// Set an alarm condition on the positive edge
IF (m_underRangeP.Q) THEN
	
	// Set underrange alarm TRUE
	Fault(fault:= f_FaultCode(TFaultPriority.Error, TFaultCondition.UnderRange), state:= TRUE);
	
END_IF
	
// Clear the alarm condition on a negative edge
IF (m_underRangeN.Q) THEN

	// Set underrange alarm FALSE
	Fault(fault:= f_FaultCode(TFaultPriority.Error, TFaultCondition.UnderRange), state:= FALSE);

END_IF

//
// Over range fault detection
//

// Use a TON delay timer
m_overRangeTON(IN:= channel.overRange);

// Rising Edge Trigger
m_overRangeP(CLK:= m_overRangeTON.Q);

// Falling Edge Trigger
m_overRangeN(CLK:= m_overRangeTON.Q);

// Set an alarm condition on the positive edge
IF (m_overRangeP.Q) THEN

	// Set overrange alarm TRUE
	Fault(fault:= f_FaultCode(TFaultPriority.Error, TFaultCondition.OverRange), state:= TRUE);
	
END_IF

// Clear the alarm condition on a negative edge
IF (m_overRangeN.Q) THEN

	// Set overrange alarm FALSE
	Fault(fault:= f_FaultCode(TFaultPriority.Error, TFaultCondition.OverRange), state:= FALSE);;
	
END_IF

//
// Short Circuit fault detection
//

// Use a TON delay timer
m_shortCircuitTON(IN:= channel.shortCircuit);

// Rising Edge Trigger
m_shortCircuitP(CLK:= m_shortCircuitTON.Q);

// Falling Edge Trigger
m_shortCircuitN(CLK:= m_shortCircuitTON.Q);

// Set an alarm condition on the positive edge
IF (m_shortCircuitP.Q) THEN

	// Set short circuit alarm TRUE
	Fault(fault:= f_FaultCode(TFaultPriority.Error, TFaultCondition.ShortCircuit), state:= TRUE);
	
END_IF

// Clear the alarm condition on a negative edge
IF (m_shortCircuitN.Q) THEN

	// Set short circuit alarm FALSE
	Fault(fault:= f_FaultCode(TFaultPriority.Error, TFaultCondition.ShortCircuit), state:= FALSE);;
	
END_IF

//
// Hardware error (wire break)
//

// Use a TON delay timer
m_errorTON(IN:= channel.error);

// Rising Edge Trigger
m_errorP(CLK:= m_errorTON.Q);

// Falling Edge Trigger
m_errorN(CLK:= m_errorTON.Q);

// Set an alarm condition on the positive edge
IF (m_errorP.Q) THEN

	// Set error alarm TRUE
	Fault(fault:= f_FaultCode(TFaultPriority.Error, TFaultCondition.HwError), state:= TRUE);
	m_WireBreakDetected := TRUE;
END_IF

// Clear the alarm condition on a negative edge
IF (m_errorN.Q) THEN

	// Set error alarm FALSE
	Fault(fault:= f_FaultCode(TFaultPriority.Error, TFaultCondition.HwError), state:= FALSE);
	m_WireBreakDetected := FALSE;
END_IF

IF (m_zeroCalEnable) THEN	

	// Calibration handling (zeroing) <TODO>
	m_zeroCalTimer();

	// Check if we are currently zeroing the transducer
	IF (m_zeroCalTimer.uliElapsedTime > 0) THEN

		// Update the data values
		m_zeroCalAccumulator := m_zeroCalAccumulator + m_filter.filteredValue;
		m_zeroCalCounter := m_zeroCalCounter + 1;

	ELSE

		// Done, calculate the average value
		IF (m_zeroCalCounter > 0) THEN

			m_rawVal := m_zeroCalAccumulator / m_zeroCalCounter;
	
		ELSE
	
			m_rawVal := m_filter.filteredValue;

		END_IF
		
		m_zeroCalRunning := FALSE;
		
	END_IF

ELSE
	
	// If no calibration is done set value to 0
	m_rawVal := 0;

END_IF

// Scale the raw calibration value to an output value
zeroCalValue := GetZeroCalValue();

(* ---------------------------------------------------------------------------
Func name   : 	AbortCal
Description : 	Aborts the calibration routine
Inputs      :	None
Returns     : 	None
Notes       : 	This routine will 0 out any previous output calibration value
--------------------------------------------------------------------------- *)

METHOD AbortCal
VAR_INPUT
END_VAR
m_zeroCalEnable := FALSE;
m_zeroCalAccumulator := 0.0;
m_zeroCalCounter := 0;
zeroCalValue := 0;
END_METHOD

(* ---------------------------------------------------------------------------
Func name   : 	Arm
Description : 	Enables all assiciated transducer alarms
Inputs      :	devId	-	device Id associated with the alarms in the system
Returns     : 	None
Notes       : 	The local alarm handler pointer is simply points to the
				global alarm handle function block.  Another approach could
				be to have any users of the analog transducer supply a
				fault handling routine with a common interface.
--------------------------------------------------------------------------- *)

METHOD Arm
VAR_INPUT
	devId		: UDeviceId;
END_VAR
// Set the local alarm handler pointer to the global handler so that the fault handler function can set alarms
m_pAlarmHandler := ADR(gAlarmHandler);

// Set the Device Id
m_devId := devId;
END_METHOD

(* ---------------------------------------------------------------------------
Func name   : 	Disarm
Description : 	Disables all assiciated transducer alarms
Inputs      :	None
Returns     : 	None
Notes       : 	This routine will also clear any active alarms before
				disabling the handler.
--------------------------------------------------------------------------- *)

METHOD Disarm
VAR_INPUT
END_VAR
// Clear any active alarms - Is this needed?
Fault(fault:= f_FaultCode(TFaultPriority.Error, TFaultCondition.UnderRange), state:= FALSE);
Fault(fault:= f_FaultCode(TFaultPriority.Error, TFaultCondition.OverRange), state:= FALSE);
Fault(fault:= f_FaultCode(TFaultPriority.Error, TFaultCondition.HwError), state:= FALSE);

// Clear the local alarm handler pointer - This will ignore all calls
m_pAlarmHandler := 0;
END_METHOD

(* ---------------------------------------------------------------------------
Func name   : 	Fault
Description : 	fault handling routine used as a common interface for
				setting/clearing transcuer faults.
Inputs      :	fault	-	fault code
				state	-	state of the fault
Returns     : 	None
Notes       : 	This routine assumes that when the transducer is armed,
				the alarm handler pointer will be non-zero, as well the
				internal m_devId parameter is set and valid.
--------------------------------------------------------------------------- *)

METHOD Fault
VAR_INPUT
	fault	: UFaultCode;
	state	: BOOL;
END_VAR
IF (m_pAlarmHandler <> 0) THEN
	
	IF (state) THEN
	
		m_pAlarmHandler^.Set(code:= f_AlarmCode(m_devId, fault));	
	
	ELSE
		
		m_pAlarmHandler^.Clear(code:= f_AlarmCode(m_devId, fault));	
	
	END_IF

END_IF
END_METHOD

(* ---------------------------------------------------------------------------
Func name   : 	FB_exit
Description : 	Destructor
Inputs      :	None
Returns     : 	None
Notes       : 	
--------------------------------------------------------------------------- *)

METHOD FB_exit : BOOL
VAR_INPUT
	bInCopyCode : BOOL; // if TRUE, the exit method is called for exiting an instance that is copied afterwards (online change)
END_VAR
// Do nothing
END_METHOD

(* ---------------------------------------------------------------------------
Func name   : 	FB_init
Description : 	Constructor
Inputs      :	iMinInput			:	minimum input
				iMaxInput			: 	maximum input
				rMinOutput			:	minimum output
				rMaxOutput			:	maximum output
				uiFilterSize 		:	Filter Sample Size
				uiFilterPrecision	:	Filter precision
				tDelay				:	Timer On Delay value
Returns     : 	None
Notes       : 	
--------------------------------------------------------------------------- *)

METHOD FB_init : BOOL
VAR_INPUT
	bInitRetains 				: BOOL; 		// if TRUE, the retain variables are initialized (warm start / cold start)
    bInCopyCode  				: BOOL; 		// if TRUE, the instance afterwards gets moved into the copy code (online change)
	iMinInput					: INT;			// minimum input
	iMaxInput					: INT;			// maximum input
	rMinOutput					: REAL;			// minimum output
	rMaxOutput					: REAL;			// maximum output
	uiFilterSize 				: UINT := 10;	// filter Sample Size
	uiFilterPrecision			: UINT := 4;	// filter precision
	tDelay						: TIME := T#1S;	// timer On Delay Value
END_VAR
// Set the member variables
m_iMinInput 	:= iMinInput;
m_iMaxInput		:= iMaxInput;
m_rMinOutput	:= rMinOutput;
m_rMaxOutput 	:= rMaxOutput;

// Initialize the calibration variables
m_zeroCalTimer.Initialize(msec:= 0, countDown:= TRUE, freeze:= FALSE);
m_zeroCalEnable := FALSE;
m_zeroCalRunning := FALSE;
m_zeroCalAccumulator := 0.0;
m_zeroCalCounter := 0;

// Initialize all of the timer delays
m_underRangeTON(PT:= tDelay);
m_overRangeTON(PT:= tDelay);
m_errorTON(PT:= tDelay);

// Initialize the Filter
// Set to default values here
m_filter.initialize(sampleSize:= uiFilterSize, precision:= uiFilterPrecision);

// Initialize the 'underrange', 'overrange', and 'error' positive edge detect signals
// to low so that we detect a positive edge if the signal is high at startup.
m_underRangeP(CLK:=FALSE);
m_overRangeP(CLK:=FALSE);
m_errorP(CLK:=FALSE);

// Initialize the output variables
signalValue := 0;
rawValue := 0;
zeroCalValue := 0;

// Set the local alarm handler pointer to the global handler
m_pAlarmHandler := ADR(gAlarmHandler);
END_METHOD

(* ---------------------------------------------------------------------------
Func name   : 	GetDevId
Description : 	Returns the transducer Device Id used for alarm categorization.
Inputs      :	None
Returns     : 	UDeviceId	-	Transducer device ID variable
Notes       : 	This function is currently used by the ENDP_Analog function block.
				I believe the End Point should set the Device Id instead of getting
				it from the transducer.  This could be a future improvement.
--------------------------------------------------------------------------- *)

METHOD GetDevId : UDeviceId
VAR_INPUT
END_VAR
GetDevId := m_devId;
END_METHOD

(* ---------------------------------------------------------------------------
Func name   : 	GetMaxOutput
Description : 	Returns the maximum output value of the transducer.
Inputs      :	None
Returns     : 	REAL	-	transducer maximum output value
Notes       : 	This routine is used by the fb_ENDP_Analog to get the
				transducer output limits.
--------------------------------------------------------------------------- *)

METHOD PUBLIC GetMaxOutput : REAL
VAR_INPUT
END_VAR
GetMaxOutput := m_rMaxOutput;
END_METHOD

(* ---------------------------------------------------------------------------
Func name   : 	GetMinOutput
Description : 	Returns the minimum output value of the transducer.
Inputs      :	None
Returns     : 	REAL	-	transducer minimum output value
Notes       : 	This routine is used by the fb_ENDP_Analog to get the
				transducer output limits.
--------------------------------------------------------------------------- *)

METHOD PUBLIC GetMinOutput : REAL
VAR_INPUT
END_VAR
GetMinOutput := m_rMinOutput;
END_METHOD

(* ---------------------------------------------------------------------------
Func name   : 	GetWireBreakStatus
Description : 	Returns the Status of a Wire Break Error.
Inputs      :	None
Returns     : 	BOOL- Status of Wire Break
Notes       : 	This method is used to get the status of the bool that reacts to a wire break.
--------------------------------------------------------------------------- *)
METHOD GetWireBreakStatus : BOOL
VAR_INPUT
END_VAR
GetWireBreakStatus := m_WireBreakDetected;
END_METHOD

(* ---------------------------------------------------------------------------
Func name   : 	GetZeroCalValue
Description : 	Scales and returns the current calibration value in mA.
Inputs      :	None
Returns     : 	REAL	-	scaled calibration value (mA)
Notes       : 	
--------------------------------------------------------------------------- *)

METHOD GetZeroCalValue : REAL
VAR_INPUT
END_VAR
// Scale the raw calibration value to an output value
 GetZeroCalValue := (m_rawVal * (m_rMaxOutput - m_rMinOutput) / (m_iMaxInput - m_iMinInput) + m_rMinOutput);
END_METHOD

(* ---------------------------------------------------------------------------
Func name   : 	InitAlarms
Description : 	Initializes the deviceId member variable used to set/clear
				the approproate alarms.
Inputs      :	devId	:	Device Id used for alarm integration
Returns     : 	None
Notes       : 	
--------------------------------------------------------------------------- *)

METHOD InitAlarms
VAR_INPUT
	devId		: UDeviceId;	// Device Id used for alarm integration
END_VAR
// Set the device id which is used for alarm integrtion
m_devId := devId;

// Register the handled alarm codes
m_pAlarmHandler^.RegisterAlarmCode(f_AlarmCode(m_devId, f_FaultCode(TFaultPriority.Error, TFaultCondition.UnderRange)));
m_pAlarmHandler^.RegisterAlarmCode(f_AlarmCode(m_devId, f_FaultCode(TFaultPriority.Error, TFaultCondition.OverRange)));
m_pAlarmHandler^.RegisterAlarmCode(f_AlarmCode(m_devId, f_FaultCode(TFaultPriority.Error, TFaultCondition.ShortCircuit)));
m_pAlarmHandler^.RegisterAlarmCode(f_AlarmCode(m_devId, f_FaultCode(TFaultPriority.Error, TFaultCondition.HwError)));
END_METHOD

(* ---------------------------------------------------------------------------
Func name   : 	IsZeroCalRunning
Description : 	Returns the status of the zero cal routine.
Inputs      :	None
Returns     : 	TRUE if zero cal running, FALSE otherwise
Notes       : 	
--------------------------------------------------------------------------- *)

METHOD IsZeroCalRunning : BOOL
VAR_INPUT
END_VAR
IsZeroCalRunning := m_zeroCalRunning;
END_METHOD

(* ---------------------------------------------------------------------------
Func name   : 	ZeroCal
Description : 	Averages the transducer signal input value to provide
				a calibration value reresenting a zero offset
Inputs      :	duration_ms	-	Duration of value averaging time in ms
Returns     : 	None
Notes       : 	This initializes the timer which runs the averaging routine
				in the main function block instantiation code.
--------------------------------------------------------------------------- *)

METHOD ZeroCal
VAR_INPUT
	duration_ms		: UINT;
END_VAR
// Initialize the data
m_zeroCalTimer.Initialize(msec := duration_ms, countDown := TRUE, freeze := FALSE);
m_zeroCalEnable := true;
m_zeroCalAccumulator := 0.0;
m_zeroCalCounter := 0;
zeroCalValue := 0;
m_zeroCalRunning := TRUE;
END_METHOD

END_FUNCTION_BLOCK

// 20 Program Organization Units/Input-Output Functions/fb_FreqTransducer
(*UPDATE: 			March. 18 2021 - Jaison Schaab

					Code Ported from Wago.
					
					Code has NOT Yet been tested.
*)

(*UPDATE: 			April. 28 2020 - Jaison Schaab

					Added the InitAlarms function which now NEEDS to be called in order to properly hook up the alarm monitors.
					This method is required because codesys does NOT properly propogate the FB_Init information like constructors
					in C code, so it is impossible to pass down the devceId information.
*)

FUNCTION_BLOCK fb_FreqTransducer
VAR_INPUT
	channel : Freq_ChannelInput; // will ~probably~ come from gstInputs. Ie HwRead + 2 copies already incurred. 
END_VAR
VAR_OUTPUT
	freqValue				: REAL;				// Scaled Signal Value (ex. mA or VDC)
	rawValue				: REAL;				// Raw Input Value (May be removed), no need to keep it UDINT, REAL is 3.4028e+38
END_VAR
VAR
	m_filter : fb_FilterExp;
	// these 2 are for Fault-handling. (hw-underrange, hw-overrange, hw-error) in this case. Which is not mapped like the Analog420input.
	m_devId : UDeviceId;
	m_pAlarmHandler : POINTER TO fb_AlarmHandler; // Alarm handler function pointer. NOTE_ Large Function. Expect this to be 1 Global func.
END_VAR

rawValue := DINT_TO_REAL(channel.value);
m_filter(inputValue:= (rawValue / 1000), filteredValue=> freqValue);

(* ---------------------------------------------------------------------------
Func name   : 	Fault
Description : 	fault handling routine used as a common interface for
				setting/clearing transcuer faults.
Inputs      :	fault	-	fault code
				state	-	state of the fault
Returns     : 	None
Notes       : 	This routine assumes that when the transducer is armed,
				the alarm handler pointer will be non-zero, as well the
				internal m_devId parameter is set and valid.
--------------------------------------------------------------------------- *)

METHOD FaultHandlerSetOrClear
VAR_INPUT
	fault	: UFaultCode;
	state	: BOOL;
END_VAR
IF (m_pAlarmHandler <> 0) THEN
	
	IF (state) THEN
	
		m_pAlarmHandler^.Set(code:= f_AlarmCode(m_devId, fault));	
	
	ELSE
		
		m_pAlarmHandler^.Clear(code:= f_AlarmCode(m_devId, fault));	
	
	END_IF

END_IF
END_METHOD

(* ---------------------------------------------------------------------------
Func name   : 	FB_init
Description : 	Constructor
Inputs      :	None
Returns     : 	None
Notes       : 	
--------------------------------------------------------------------------- *)

METHOD FB_init : BOOL
VAR_INPUT
	bInitRetains 		: BOOL; 		// if TRUE, the retain variables are initialized (warm start / cold start)
    bInCopyCode  		: BOOL; 		// if TRUE, the instance afterwards gets moved into the copy code (online change)
	histavgFiltSize: UINT;
	histavgFiltPrecision: UINT;
END_VAR
m_filter.initialize(sampleSize:= histavgFiltSize, precision:= histavgFiltPrecision);
freqValue := 0;
rawValue := 0;
END_METHOD

METHOD GetDevId : UDeviceId
VAR_INPUT
END_VAR
GetDevId := m_devId;
END_METHOD

(* ---------------------------------------------------------------------------
Func name   : 	InitAlarms
Description : 	Initializes the deviceId member variable used to set/clear
				the approproate alarms.
Inputs      :	devId	:	Device Id used for alarm integration
Returns     : 	None
Notes       : 	
--------------------------------------------------------------------------- *)

METHOD InitAlarms
VAR_INPUT
	devId : UDeviceId;
END_VAR
// Set the device id which is used for alarm integrtion
m_devId := devId;

// Register the handled alarm codes
// None Defined Yet <JAISON>
END_METHOD

END_FUNCTION_BLOCK

// 20 Program Organization Units/Instrument-Controller Functions/fb_Densitometer
(*AUTHOR:			Ryan Herdian*)
(*DATE:				June 16 / 2020*)
(*DESCRIPTION: 		This Function Block provides a BASE class for all densitometer objects.  The class
					consists of the following features:
					
						-	Min/Max configurable density ranges in specific gravity units whose range/values define the density units 
							of the entire class. Density is ratio agains clean water. Specific gravity of 1 is clean water.
						-	Raw density value in specific gravity units which is to be set by the derived class from its data source
						-	User settable unitless k-factor value which allows corrections in the desnsity value
						-	Corrected density value in density units which is the raw flow with k-factor applied
						-	Automatic k-factor calculation given known reference density in density units
					
					No Alarms are currently included, however alarm handler / fault function are defined.*)

(*NOTES:			The derived densitometer class is required to:
					
						- 	Set the m_densityMin/m_densityMax values in density unit [SGU].
							For example if the range of (0 - 1 [SGU]) then all values in that densitometer / denso instance
							 will return values in Specific Gravity Unit.  Including raw/corrected density.
						-	Set the m_rawDensity value in density units using the SetRawFlow() method.
						-	Initialize all values in the constructor including the user k-factor 
							and setting the alarm handler pointer.

*)

(*UPDATE: 			March. 18 2021 - Jaison Schaab

					Code Ported from Wago.
					
					Code has NOT Yet been tested.
*)

FUNCTION_BLOCK fb_Densitometer
VAR_INPUT
END_VAR
VAR_OUTPUT
END_VAR
VAR
	m_densityMin		: REAL			:= 0.0;			// in Specific Gravity Unit [SGU]
	m_densityMax		: REAL			:= 0.0;			// in [SGU]
	
	m_rawDensity		: REAL			:= 0.0;			// in density unit, e.g.: [SGU]
	
	m_userkfact			: REAL			:= 1.0;			// unitless multiplier (1.0 simply allows raw value output)
	
	// Fault Handling (Alarms)
	m_devId				: UDeviceId;					// Device Id used for alarm integration
END_VAR
VAR CONSTANT
	USER_K_FACTOR_MIN	: REAL := 0.1;					// minimum allowable user k-factor
	USER_K_FACTOR_MAX	: REAL := 10.0;					// maximum allowable user k-factor		
END_VAR

(* ---------------------------------------------------------------------------
Func name   : 	CalculateUserKFact
Description : 	Routine will calculate and set the densitometer k-factor
				so that the corrected density matches the input reference
				density value.
Inputs      :	refDensity	-	reference density value in density unit [SGU]
Returns     : 	None
Notes       : 	Use this routine to calibrate the densitometer to a known
				density in [SGU].
--------------------------------------------------------------------------- *)

METHOD CalculateUserkFact
VAR_INPUT
	refDensity	: REAL;		// reference density value in density unit [SGU]
END_VAR
IF (m_rawDensity > 0.0) THEN
	setUserKFact(kfact:= (refDensity / m_rawDensity) );
END_IF
END_METHOD

(* ---------------------------------------------------------------------------
Func name   : 	GetCorrectedDensitySGU
Description : 	Routine to calculate and return the corrected density
				with the user k-factor applied in density unit [SGU].
Inputs      :	None
Returns     : 	REAL	-	The corrected density value in density unit [SGU]
Notes       : 	
--------------------------------------------------------------------------- *)

METHOD GetCorrectedDensitySGU : REAL
VAR_INPUT
END_VAR
GetCorrectedDensitySGU	:= m_userkfact * m_rawDensity;
END_METHOD

(* ---------------------------------------------------------------------------
Func name   : 	GetDensityRange_MinMax
Description : 	Gets the minimum/maximum density range values from the densitometer
				in specific gravity units. Specific gravity of 1 is clean water.
Inputs      :	None
Returns     : 	minDensity		: 	denso minimum density value in density unit [SGU]
				maxDensity		:	denso maximum density value in density unit [SGU]
Notes       : 	
--------------------------------------------------------------------------- *)

METHOD GetDensityRange_MinMax
VAR_INPUT
END_VAR
VAR_OUTPUT
	minDensity		: REAL;		// minimum density value at transducer minimum value in [SGU]
	maxDensity		: REAL;		// maximum desnity value at transducer maximum value in [SGU]
END_VAR
// output the min/max density ranges
minDensity	:= m_densityMin;		// minimum density value at transducer minimum value in density unit [SGU]
maxDensity	:= m_densityMax;		// maximum desnity value at transducer maximum value in density unit [SGU]
END_METHOD

(* ---------------------------------------------------------------------------
Func name   : 	GetRawDensity
Description : 	Routine to return the raw density in density unit [SGU].
				This value does not have the k-factor applied.
Inputs      :	None
Returns     : 	REAL	-	The raw density value in Specific in density unit [SGU]
Notes       : 	
--------------------------------------------------------------------------- *)

METHOD GetRawDensity : REAL
VAR_INPUT
END_VAR
GetRawDensity	:= m_rawDensity;
END_METHOD

(* ---------------------------------------------------------------------------
Func name   : 	GetUserKFact
Description : 	Routine will return the unitless user k-factor value.
Inputs      :	None
Returns     : 	REAL	-	The unitless user k-factor value
Notes       : 	
--------------------------------------------------------------------------- *)

METHOD GetUserKFact : REAL
VAR_INPUT
END_VAR
GetUserKFact := m_userkfact;
END_METHOD

(* ---------------------------------------------------------------------------
Func name   : 	InitAlarms
Description : 	Initializes the deviceId member variable used to set/clear
				the approproate alarms.
Inputs      :	None
Returns     : 	None
Notes       : 	
--------------------------------------------------------------------------- *)

METHOD InitAlarms
VAR_INPUT
	devId		: UDeviceId;	// Device Id used for alarm integration
END_VAR
// Set the device id which is used for alarm integrtion
m_devId := devId;
END_METHOD

(* ---------------------------------------------------------------------------
Func name   : 	SetDensityRange_MinMax
Description : 	Sets the minimum/maximum desnity range values for the densitometer / denso
				in density unit Specific Gravity, [SGU].  The units defined by this range will
				define the units for all flow meter values.
Inputs      :	minDensity		: 	densitometer minimum flow value in density unit [SGU]
				maxDensity		:	densitometer maximum flow value in density unit [SGU]
Returns     : 	TRUE if min and max density are set. 
				FALSE if min and max density are not set (min density is greater than or equal to max density).
Notes       : 	All values in densitometer instance should be interpreted as 
				Specific Gravity, [SGU], including raw/corrected density.
--------------------------------------------------------------------------- *)

METHOD SetDensityRange_MinMax	: BOOL
VAR_INPUT
	minDensity		: REAL;		// minimum density value at transducer minimum value in density unit [SGU]
	maxDensity		: REAL;		// maximum density value at transducer maximum value in density unit [SGU]
END_VAR
IF (minDensity < maxDensity) THEN

	// Set the min/max densitometer range
	m_densityMin	:= minDensity;
	m_densityMax	:= maxDensity;
	
	SetDensityRange_MinMax	:= TRUE;

ELSE
	
	SetDensityRange_MinMax	:= FALSE;

END_IF
END_METHOD

(* ---------------------------------------------------------------------------
Func name   : 	SetRawDensity
Description : 	Private function which allows the derived classes to set the 
				densitometer rawDensity value in density unit [SGU].  
Inputs      :	density	-	Raw density in density unit [SGU]
Returns     : 	None
Notes       : 	The value will be limited by the initialized 
				minDensity/maxDensity values.
--------------------------------------------------------------------------- *)

METHOD PROTECTED SetRawDensity
VAR_INPUT
	density		: REAL;		// in density unit [SGU]
END_VAR
// Set the raw density value in the base densitometer class in density unit [SGU]
m_rawDensity	:= MAX(MIN(density, m_densityMax), m_densityMin);
END_METHOD

(* ---------------------------------------------------------------------------
Func name   : 	SetUserKFact
Description : 	Routine to set the unitless user k-factor value.
Inputs      :	kfact	-	The desried unitless user k-factor value
Returns     : 	None
Notes       : 	The value will be limited by the constants 
				USER_K_FACTOR_MIN and USER_K_FACTOR_MAX.
--------------------------------------------------------------------------- *)

METHOD setUserKFact
VAR_INPUT
	kfact	: REAL;
END_VAR
m_userkfact := MAX(MIN(kfact, USER_K_FACTOR_MAX), USER_K_FACTOR_MIN);
END_METHOD

END_FUNCTION_BLOCK

// 20 Program Organization Units/Instrument-Controller Functions/fb_ENDP_AnalogCalPressure
(*UPDATE: 			March. 18 2021 - Jaison Schaab

					Code Ported from Wago.
					
					Code has NOT Yet been tested.
*)

FUNCTION_BLOCK fb_ENDP_AnalogCalPressure
VAR_INPUT
	
END_VAR
VAR_OUTPUT
	correctedPressure 		: REAL;
	endpState				: INT;
END_VAR
VAR
	//Transducer Input
	m_pTransducer 	  		: POINTER TO fb_AnalogTransducer;
	
	//Config Variables - Need Get/Set Routines
	m_lowerCalPoint	  		: TCalibrationDataPoint; // m_inMin & m_outMin
	m_upperCalPoint	  		: TCalibrationDataPoint;//  m_inMax & m_outMax
	
	//Current configured pressure limits
	m_defaultPressMin 		: REAL := 0.0;
	m_defaultPressMax 		: REAL := 0.0;
	
	m_pressureMin		  		: REAL := 0.0; // physMin
	m_pressureMax		  		: REAL := 0.0; // physMax
	
	// Vars in fb_ENDP_Analog
	m_outDiffMultiplier 		: REAL;
	m_inDiffDivisor				: REAL; 
	m_offset					: REAL;
	m_hysteresis 				: REAL;
	
	m_rawPressure				: REAL := 0.0;
	m_userkfactor 				: REAL := 0.0;
	
	
	//Internal Status
	m_lowerCalTrigger 		: R_TRIG;
	m_upperCalTrigger 		: R_TRIG;
	
	m_calibrateLowPoint 	: BOOL;
	m_calibrateHighPoint 	: BOOL;
	// Handle Alarms
	m_devId 				: UDeviceId;
	LowAlarmMonitor			: fb_AlarmMonitor;
	LowWarningMonitor		: fb_AlarmMonitor;
	HighWarningMonitor		: fb_AlarmMonitor;
	HighAlarmMonitor		: fb_AlarmMonitor;
END_VAR

VAR CONSTANT
	USER_K_FACTOR_MAX 		: REAL := 10.0;
	USER_K_FACTOR_MIN 		: REAL := 1.0;
	DELAY_TON				: TIME := T#200MS;
END_VAR

// Ensure transducer pointer is not NULL
IF (m_pTransducer <> _NULL) THEN
	
	m_lowerCalTrigger(CLK:= (NOT m_pTransducer^.IsZeroCalRunning()) AND (m_calibrateLowPoint));
 	IF (m_lowerCalTrigger.Q) THEN
		m_lowerCalPoint.xValue	:= m_pTransducer^.GetZeroCalValue();
		
		m_calibrateLowPoint := FALSE;

		// Calculate a new minimum flow
		SetPressureRange(	minimum := f_LinearScale(value		:= m_pTransducer^.GetMinOutput(), 
															minInput	:= m_lowerCalPoint.xValue, 
															maxInput	:= m_upperCalPoint.xValue, 
															minOutput	:= m_lowerCalPoint.yValue, 
															maxOutput	:= m_upperCalPoint.yValue),
							maximum	:= m_pressureMax);
	END_IF
	
	m_upperCalTrigger(CLK:= (NOT m_pTransducer^.IsZeroCalRunning()) AND (m_calibrateHighPoint));
	IF (m_upperCalTrigger.Q) THEN
		m_upperCalPoint.xValue	:= m_pTransducer^.GetZeroCalValue();
		
		m_calibrateHighPoint := FALSE;
		
		// Calculate a new maximum pressure
		SetPressureRange(	minimum := m_pressureMin,
							maximum	:= f_LinearScale(value		:= m_pTransducer^.GetMaxOutput(), 
															minInput	:= m_lowerCalPoint.xValue, 
															maxInput	:= m_upperCalPoint.xValue, 
															minOutput	:= m_lowerCalPoint.yValue, 
															maxOutput	:= m_upperCalPoint.yValue));
	END_IF
	
	IF (NOT m_pTransducer^.IsZeroCalRunning()) THEN
		SetRawPressure( pressure := f_LinearScale(	value		:= m_pTransducer^.signalValue, 
															minInput	:= m_lowerCalPoint.xValue, 
															maxInput	:= m_upperCalPoint.xValue, 
															minOutput	:= m_lowerCalPoint.yValue, 
															maxOutput	:= m_upperCalPoint.yValue));
	END_IF							
ELSE
	SetRawPressure( pressure := 0.0);
END_IF

// Output the corrected pressure Value in kpa units
correctedPressure := GetCorrectedPressure();

//Monitor alarms.
LowAlarmMonitor.MonitorReal(correctedPressure);
LowWarningMonitor.MonitorReal(correctedPressure);
HighWarningMonitor.MonitorReal(correctedPressure);
HighAlarmMonitor.MonitorReal(correctedPressure);

IF (m_pTransducer^.channel.error) THEN
	endpState := TEnuHmiGaugeState.LowAlarm;
ELSIF(LowAlarmMonitor.GetState()) THEN
	endpState := TEnuHmiGaugeState.LowAlarm;
ELSIF(HighWarningMonitor.GetState()) THEN
	endpState := TO_INT(TEnuHmiGaugeState.HighWarning);
ELSIF(LowWarningMonitor.GetState()) THEN
	endpState := TEnuHmiGaugeState.LowWarning;
ELSE
	endpState := TEnuHmiGaugeState.No_Alarm;			
END_IF

(* ---------------------------------------------------------------------------
Func name   : 	CalculateUserKFact
Description : 	
Inputs      :	
Returns     : 	None
Notes       : 	
--------------------------------------------------------------------------- *)

METHOD CalculateUserKFactor
VAR_INPUT
	refPress	: REAL;
END_VAR
IF (m_rawPressure > 0.0) THEN
	SetUserKFactor(refPress  / m_rawPressure);
END_IF
END_METHOD

(* ---------------------------------------------------------------------------
Func name   : 	CalibrateHighDataPoint
Description : 	Averages the transducer signal input value to provide
				a high calibration data point for the flowmeter scale.
Inputs      :	val			-	Calibration value in Kpa units
				duration_ms	-	Duration of value averaging time in ms
Returns     : 	None
Notes       : 	
--------------------------------------------------------------------------- *)

METHOD CalibrateHighDataPoint
VAR_INPUT
	val				: REAL;		// Calibration value in volume/t units
	duration_ms 	: UINT;		// Duration of value averaging time in ms
END_VAR
IF ((NOT m_calibrateLowPoint) AND (NOT m_calibrateHighPoint)) THEN
	m_pTransducer^.ZeroCal(duration_ms:= duration_ms);
	m_upperCalPoint.yValue	:= val;
	m_calibrateHighPoint := TRUE;
END_IF
END_METHOD

(* ---------------------------------------------------------------------------
Func name   : 	CalibrateLowDataPoint
Description : 	Averages the transducer signal input value to provide
				a low calibration data point for the flowmeter scale.
Inputs      :	val			-	Calibration value in volume/t units
				duration_ms	-	Duration of value averaging time in ms
Returns     : 	None
Notes       : 	
--------------------------------------------------------------------------- *)

METHOD CalibrateLowDataPoint
VAR_INPUT
	val				: REAL;		// Calibration value in volume/t units
	duration_ms 	: UINT;		// Duration of value averaging time in ms
END_VAR
VAR
	minFlow		: REAL;
	maxFlow		: REAL;
END_VAR
IF ((NOT m_calibrateLowPoint) AND (NOT m_calibrateHighPoint)) THEN
	m_pTransducer^.ZeroCal(duration_ms:= duration_ms);
	m_lowerCalPoint.yValue	:= val;
	m_calibrateLowPoint := TRUE;
END_IF
END_METHOD

(* ---------------------------------------------------------------------------
Func name   : 	ClearCalibration
Description : 	Clears all calibration of the pressure transducer and resets to
				the default constructor scale.
Inputs      :	None
Returns     : 	None
Notes       : 	
--------------------------------------------------------------------------- *)

METHOD ClearCalibration
VAR_INPUT
END_VAR
// Reset to default values
m_lowerCalPoint.xValue	:= m_pTransducer^.GetMinOutput();
m_lowerCalPoint.yValue	:= m_defaultPressMin;

m_upperCalPoint.xValue	:= m_pTransducer^.GetMaxOutput();
m_upperCalPoint.yValue	:= m_defaultPressMax;

SetPressureRange(minimum := m_defaultPressMin,maximum := m_defaultPressMax);
						
m_calibrateLowPoint		:= FALSE;
m_calibrateHighPoint	:= FALSE;
END_METHOD

(* ---------------------------------------------------------------------------
Func name   : 	FB_exit
Description : 	Destructor
Inputs      :	None
Returns     : 	None
Notes       : 	
--------------------------------------------------------------------------- *)

METHOD FB_exit : BOOL
VAR_INPUT
	bInCopyCode : BOOL; // if TRUE, the exit method is called for exiting an instance that is copied afterwards (online change)
END_VAR
// Do nothing
END_METHOD

METHOD FB_Init
VAR_INPUT
	bInitRetains 	: BOOL;
	bInCopyCode  	: BOOL;
	
	pTransducer  	: POINTER TO fb_AnalogTransducer;
	minPress	 	: REAL;
	maxPress	 	: REAL;
	perctHysteresis : REAL;
END_VAR
// Default User K-Factor to 1.0
SetUserKFactor( k := 1.0);

// Default the raw press value to 0
SetRawPressure( pressure := 0.0);

// Set the pressure ranges in pascals
m_defaultPressMin := minPress;
m_defaultPressMax := maxPress;

SetPressureRange( minimum := minPress, maximum := maxPress);

// Set the transducer pointer
m_pTransducer := pTransducer;

// Initialize the calibration values
m_lowerCalPoint.xValue := m_pTransducer^.GetMinOutput(); //inMin
m_lowerCalPoint.yValue := minPress; //outMin

m_upperCalPoint.xValue := m_pTransducer^.GetMaxOutput(); // inMax
m_upperCalPoint.yValue := maxPress; // outMax

m_outDiffMultiplier    := m_upperCalPoint.yValue - m_lowerCalPoint.yValue;
m_inDiffDivisor		   := m_upperCalPoint.xValue - m_upperCalPoint.xValue;

IF( m_inDiffDivisor = 0.0) THEN
	m_inDiffDivisor := 0.000001; //protect against div-by-0, only ONCE, and produce VERY-LARGE Bad value.
                                  //Beckhoff-tcNov was doing this A.every cycle and B.returned 0.0 if Bad, which is normal value. hard to notice.
END_IF


m_hysteresis := perctHysteresis / 100;
m_lowerCalTrigger(CLK := FALSE);
m_upperCalTrigger(CLK := FALSE);

m_calibrateLowPoint 	:= FALSE;
m_calibrateHighPoint 	:= FALSE;
END_METHOD

(* ---------------------------------------------------------------------------
Func name   : 	GetConfigData
Description : 	equivalent of "Configure" bkhff-legacy-names.
				
Inputs      :	2-end-range-values, 1 offset, 4 alarms - 7 values.
				state	-	state of the fault
Returns     : 	None
Notes       : 	
--------------------------------------------------------------------------- *)

METHOD GetConfigData
VAR_INPUT
	//cfg : TEndpAnalogCfg;
MinValue : REAL;
MaxValue : REAL;
OffsetValue : REAL;
LowLimit : REAL;
LowWarning : REAL;
HighWarning : REAL;
HighLimit : REAL;
END_VAR
m_lowerCalPoint.yValue := MinValue;
m_upperCalPoint.yValue := MaxValue;
m_offset := OffsetValue;

//LowAlarmMonitor.m_limit.limitOn := LowLimit;
LowAlarmMonitor.SetLimitReal(LowLimit, LowLimit*(1 + m_hysteresis)); // + 0.5);

//LowWarningMonitor.m_limit.limitOn := LowWarning;
LowWarningMonitor.SetLimitReal(LowWarning, LowWarning*(1 + m_hysteresis)); // + 0.5);

//HighWarningMonitor.m_limit.limitOn := HighWarning;
HighWarningMonitor.SetLimitReal(HighWarning, HighWarning*(1 - m_hysteresis)); // - 0.5);

//HighAlarmMonitor.m_limit.limitOn := HighLimit;
HighAlarmMonitor.SetLimitReal(HighLimit, HighLimit*(1 - m_hysteresis)); // - 0.5);
END_METHOD

METHOD GetCorrectedPressure : REAL
VAR_INPUT
END_VAR
GetCorrectedPressure := m_userkfactor * m_rawPressure;
END_METHOD

(* ---------------------------------------------------------------------------
Func name   : 	GetLowerCalDataPoint
Description : 	returns the flowmeter lower calibration data point.
Inputs      :	None
Returns     : 	REAL	-	lower calibration data point
Notes       : 	
--------------------------------------------------------------------------- *)

METHOD GetLowerCalDataPoint : TCalibrationDataPoint
VAR_INPUT
END_VAR
GetLowerCalDataPoint := m_lowerCalPoint;
END_METHOD

(* ---------------------------------------------------------------------------
Func name   : 	GetPressureRange
Description : 	Gets the minimum/maximum pressure range values from the pressure transducer
				in volume/t units.
Inputs      :	None
Returns     : 	minPressure		: 	Pressure Transducer's minimum pressure value (kpa)
				maxPressure		:	Pressure Transducer's maximum pressure value (kpa)
Notes       : 	
--------------------------------------------------------------------------- *)

METHOD GetPressureRange
VAR_INPUT
END_VAR
VAR_OUTPUT
	minPressure : REAL;	// minimum pressure value at transducer's minimum value (kpa)
	maxPressure : REAL; // maximum pressure value at transducer's maximum value (kpa)
END_VAR
minPressure := m_pressureMin;
maxPressure := m_pressureMax;
END_METHOD

(* ---------------------------------------------------------------------------
Func name   : 	GetRawPressure
Description : 	Routine to return the raw pressure value in Kpa units.
				This value does not have the k-factor applied.
Inputs      :	None
Returns     : 	REAL	-	The raw pressure value in Kpa
Notes       : 	
--------------------------------------------------------------------------- *)

METHOD GetRawPressure : REAL
VAR_INPUT
END_VAR
GetRawPressure := m_rawPressure;
END_METHOD

(* ---------------------------------------------------------------------------
Func name   : 	GetUpperCalDataPoint
Description : 	returns the flowmeter upper calibration data point.
Inputs      :	None
Returns     : 	REAL	-	upper calibration data point
Notes       : 	
--------------------------------------------------------------------------- *)

METHOD GetUpperCalDataPoint : TCalibrationDataPoint
VAR_INPUT
END_VAR
GetUpperCalDataPoint := m_upperCalPoint;
END_METHOD

METHOD GetUserAlarms
VAR_OUTPUT
	outLAlarm 	:REAL;
	outLWarn 	:REAL;
	outHWarn 	:REAL;
	outHAlarm 	:REAL;
END_VAR
outLAlarm 	:= LREAL_TO_REAL(LowAlarmMonitor.m_limit.limitOn);
outLWarn  	:= LREAL_TO_REAL(LowWarningMonitor.m_limit.limitOn);
outHWarn 	:= LREAL_TO_REAL(HighWarningMonitor.m_limit.limitOn);
outHAlarm 	:= LREAL_TO_REAL(HighAlarmMonitor.m_limit.limitOn);
END_METHOD

(* ---------------------------------------------------------------------------
Func name   : 	GetUserKFactor
Description : 	Routine will return the unitless user k-factor value.
Inputs      :	None
Returns     : 	REAL	-	The unitless user k-factor value
Notes       : 	
--------------------------------------------------------------------------- *)

METHOD GetUserKFactor : REAL
VAR_INPUT
END_VAR
GetUserKFactor := m_userkfactor;
END_METHOD

(* ---------------------------------------------------------------------------
Func name   : 	InitAlarms
Description : 	Initializes the deviceId member variable used to set/clear
				the approproate alarms.
Inputs      :	None
Returns     : 	None
Notes       : 	
--------------------------------------------------------------------------- *)

METHOD InitAlarms
VAR_INPUT
END_VAR
// Set the device id which is used for alarm integration
m_devId := m_pTransducer^.GetDevId();

LowAlarmMonitor.InitAlarm(f_AlarmCode(m_devId, f_FaultCode(TFaultPriority.Warning, TFaultCondition.UnderLimit)), TAlarmMonitorType.lower_limit, DELAY_TON);
LowWarningMonitor.InitAlarm(f_AlarmCode(m_devId, f_FaultCode(TFaultPriority.Warning, TFaultCondition.UnderWarning)), TAlarmMonitorType.lower_limit, DELAY_TON);
HighWarningMonitor.InitAlarm(f_AlarmCode(m_devId, f_FaultCode(TFaultPriority.Warning, TFaultCondition.OverWarning)), TAlarmMonitorType.upper_limit, DELAY_TON);
HighAlarmMonitor.InitAlarm(f_AlarmCode(m_devId, f_FaultCode(TFaultPriority.Warning, TFaultCondition.OverLimit)), TAlarmMonitorType.upper_limit, DELAY_TON);
END_METHOD

METHOD SetHysteresis
VAR_INPUT
	perctHysteresis : REAL;
END_VAR
m_hysteresis := perctHysteresis/100;
END_METHOD

(* ---------------------------------------------------------------------------
Func name   : 	SetLowerCalDataPoint
Description : 	sets the flowmeter lower calibration data point.
Inputs      :	calPoint	-	calibration data point
Returns     : 	None
Notes       : 	
--------------------------------------------------------------------------- *)

METHOD SetLowerCalDataPoint
VAR_INPUT
	calPoint	: TCalibrationDataPoint;
END_VAR
m_lowerCalPoint := calPoint;
END_METHOD

METHOD SetPressureRange : BOOL
VAR_INPUT
	minimum : REAL;
	maximum : REAL;
END_VAR
IF ( maximum > minimum) THEN
	m_pressureMin := minimum;
	m_pressureMax := maximum;
	SetPressureRange := TRUE;
ELSE
	SetPressureRange := FALSE;
END_IF
END_METHOD

METHOD SetRangeUserAlarms
VAR_INPUT
	loAlarm : REAL;
	loWarn  : REAL;
	hiWarn  : REAL;
	hiAlarm : REAL;
END_VAR
IF (NOTUSED = loAlarm OR NOTUSED_LOMAX = loAlarm OR loAlarm < m_lowerCalPoint.yValue OR loAlarm > m_upperCalPoint.yValue) THEN
	loAlarm := NOTUSED_LOMAX;
	LowAlarmMonitor.DisableLimit();
ELSE
	LowAlarmMonitor.EnableLimit();
END_IF
LowAlarmMonitor.SetLimitReal(loAlarm, (loAlarm  + MAX(0.001, ABS(loAlarm)) * m_hysteresis));

IF (NOTUSED = loWarn OR loWarn <= loAlarm OR loAlarm > m_upperCalPoint.yValue ) THEN
	loWarn := loAlarm;
	LowWarningMonitor.DisableLimit();
ELSE
	LowWarningMonitor.EnableLimit();
END_IF
LowWarningMonitor.SetLimitReal(loWarn, (loWarn  + MAX(0.001, ABS(loWarn)) * m_hysteresis));

IF (NOTUSED = hiAlarm OR NOTUSED_HIMAX = hiAlarm OR hiAlarm < m_lowerCalPoint.yValue OR hiAlarm > m_upperCalPoint.yValue) THEN
	hiAlarm := NOTUSED_HIMAX; //Guaranteed greater than m_outMax; We pick _some_ large value.
	HighAlarmMonitor.DisableLimit();
ELSE
	HighAlarmMonitor.EnableLimit();
END_IF
HighAlarmMonitor.SetLimitReal(hiAlarm, (hiAlarm - MAX(0.001, ABS(hiAlarm)) * m_hysteresis));

IF (NOTUSED = hiWarn OR hiWarn >= hiAlarm OR hiWarn < m_lowerCalPoint.yValue) THEN
	hiWarn := hiAlarm;   //User doesnt have ability to set these individually. So WE define this order. So hiAlarm - already set.
	HighWarningMonitor.DisableLimit();
ELSE
	HighWarningMonitor.EnableLimit();
END_IF
HighWarningMonitor.SetLimitReal(hiWarn, (hiWarn - MAX(0.001, ABS(hiWarn)) * m_hysteresis));
END_METHOD

METHOD SetRawPressure : REAL
VAR_INPUT
	pressure : REAL;
END_VAR
m_rawPressure := MAX(MIN(pressure,m_pressureMax), m_pressureMin);

SetRawPressure := m_rawPressure;
END_METHOD

(* ---------------------------------------------------------------------------
Func name   : 	SetUpperCalDataPoint
Description : 	sets the flowmeter upper calibration data point.
Inputs      :	calPoint	-	calibration data point
Returns     : 	None
Notes       : 	
--------------------------------------------------------------------------- *)

METHOD SetUpperCalDataPoint
VAR_INPUT
	calPoint	: TCalibrationDataPoint;
END_VAR
m_upperCalPoint := calPoint;
END_METHOD

METHOD SetUserKFactor
VAR_INPUT
	k : REAL;
END_VAR
m_userkfactor := MAX(MIN(k, USER_K_FACTOR_MAX), USER_K_FACTOR_MIN);
END_METHOD

END_FUNCTION_BLOCK

// 20 Program Organization Units/Instrument-Controller Functions/fb_ENDP_AnalogDensitometer
(*AUTHOR:			Ryan Herdian*)
(*DATE:				June 17, 2020*)
(*DESCRIPTION: 		Derived densitometer class which provides an analog denso object.  The raw density
					value is obtained from the configured "Analog Transducer" object in the configured
					density unit, Specific Gravity Unit [SGU].*)

(*UPDATE: 			March. 18 2021 - Jaison Schaab

					Code Ported from Wago.
					
					Code has NOT Yet been tested.
*)

FUNCTION_BLOCK fb_ENDP_AnalogDensitometer EXTENDS fb_Densitometer
VAR_INPUT
END_VAR
VAR_OUTPUT
	correctedDensity	: REAL;								// Corrected density in density unit Specific Gravity Unit, [SGU]
END_VAR
VAR
	// Transducer input
	m_pTransducer	 	: POINTER TO fb_AnalogTransducer;	// Pointer to transducer
END_VAR

// Ensure transducer pointer is not NULL
IF (m_pTransducer <> _NULL) THEN

	// Set the raw density value in the base densitometer class in density unit, e.g.: Specific Gravity Unit, [SGU]
	SetRawDensity(density:= f_LinearScale(	value		:= m_pTransducer^.signalValue, 
											minInput	:= m_pTransducer^.GetMinOutput(), 
											maxInput	:= m_pTransducer^.GetMaxOutput(), 
											minOutput	:= m_densityMin, 
											maxOutput	:= m_densityMax));
													
ELSE
	SetRawDensity(density:= 0.0);

END_IF
							
// Output the corrected Flow Value in voume/t units
correctedDensity := GetCorrectedDensitySGU();

(* ---------------------------------------------------------------------------
Func name   : 	FB_exit
Description : 	Destructor
Inputs      :	None
Returns     : 	None
Notes       : 	
--------------------------------------------------------------------------- *)

METHOD FB_exit : BOOL
VAR_INPUT
	bInCopyCode : BOOL; // if TRUE, the exit method is called for exiting an instance that is copied afterwards (online change)
END_VAR
// Do Nothing
END_METHOD

(* ---------------------------------------------------------------------------
Func name   : 	FB_init
Description : 	Constructor
Inputs      :	pTransducer			:	transducer pointer
				minDensity			: 	minimum density value at transducer minimum value in density unit, e.g.: Specific Gravity Unit, [SGU]
				maxDensity			:	maximum density value at transducer maximum value in density unit, e.g.: Specific Gravity Unit, [SGU]
Returns     : 	None
Notes       : 	
--------------------------------------------------------------------------- *)

METHOD FB_init : BOOL
VAR_INPUT
	bInitRetains 		: BOOL; 							// if TRUE, the retain variables are initialized (warm start / cold start)
    bInCopyCode  		: BOOL; 							// if TRUE, the instance afterwards gets moved into the copy code (online change)
	pTransducer 		: POINTER TO fb_AnalogTransducer;	// transducer pointer
	minDensity 			: REAL;								// minimum Density value at transducer minimum value in density unit, e.g.: Specific Gravity Unit, [SGU]
	maxDensity 			: REAL;								// maximum Density value at transducer maximum value in density unit, e.g.: Specific Gravity Unit, [SGU]
END_VAR
// Default User kFact to 1.0
SetUserKFact(kfact := 1.0);

// Default the raw density value to 0
SetRawDensity(density:= 0.0);

// Set the density ranges in density unit, e.g.: Specific Gravity Unit, [SGU]
SetDensityRange_MinMax(	minDensity	:= minDensity, 
						maxDensity	:= maxDensity);

// Set the transducer pointer
m_pTransducer := pTransducer;
END_METHOD

END_FUNCTION_BLOCK

// 20 Program Organization Units/Instrument-Controller Functions/fb_ENDP_AnalogFlowmeter
(*AUTHOR:			Jaison Schaab*)
(*DATE:				June 9 / 2020*)
(*DESCRIPTION: 		Derived flow meter class which provides an analog flow meter object.  The raw volume flow
					value is obtained from the configured "Analog Transducer" object in the configured
					 volume/t units.*)

(*UPDATE: 			March. 23 2021 - Jaison Schaab

					Code Is fully tested and functional.				
*)
					 
(*UPDATE: 			March. 18 2021 - Jaison Schaab

					Code Ported from Wago.
					
					Code has NOT Yet been tested.
*)
					 
(*UPDATE: 			August. 31 2020 - Jaison Schaab

					Added new calibration data points to define the analog flow meter scaling.  These data points can
					be reset to the constructor values using the "ClearCalibration" routine.  They are set using the
					"CalibrateHighDataPoint" and "CalibrateLowDataPoint" or by simply writing them via the "SetLowerCalDataPoint"
					and "SetUpperCalDataPoint".
					
					Keep in mind that these values will need to be added to the config memory space in order to retain them.
*)	
					 
(*UPDATE: 			June. 23 2020 - Jaison Schaab

					Removed backdoor (m_pAlarmHandler : POINTER TO fb_AlarmHandler) alarm handler function pointer
					in order to simplify the alarm system.  Any alarms at this level should define a instance
					of the fb_AlarmMonitor class which will handle the alarm registration/set/clear.
*)					 				 

FUNCTION_BLOCK fb_ENDP_AnalogFlowmeter EXTENDS fb_FlowMeter
VAR_INPUT
END_VAR
VAR_OUTPUT
	correctedFlow				: REAL;								// Corrected flow in volume/t units
END_VAR
VAR
	// Transducer input
	m_pTransducer				: POINTER TO fb_AnalogTransducer;	// Pointer to transducer
	
	// Config Variables - Need Get/Set Routines
	m_lowerCalPoint				: TCalibrationDataPoint;			// Lower calibration data point
	m_upperCalPoint				: TCalibrationDataPoint;			// Upper calibration data point
	
	
	// Internal Status
	m_lowerCalTrigger			: R_TRIG;
	m_upperCalTrigger			: R_TRIG;
	
	m_calibrateLowPoint			: BOOL;
	m_calibrateHighPoint		: BOOL;

END_VAR

// Ensure transducer pointer is not NULL
IF (m_pTransducer <> _NULL) THEN
	
	m_lowerCalTrigger(CLK:= (NOT m_pTransducer^.IsZeroCalRunning()) AND (m_calibrateLowPoint));
 	IF (m_lowerCalTrigger.Q) THEN
		m_lowerCalPoint.xValue	:= m_pTransducer^.GetZeroCalValue();
		
		m_calibrateLowPoint := FALSE;

		// Calculate a new minimum flow
		SetFlowRange_MinMax(	minFlow := f_LinearScale(	value		:= m_pTransducer^.GetMinOutput(), 
															minInput	:= m_lowerCalPoint.xValue, 
															maxInput	:= m_upperCalPoint.xValue, 
															minOutput	:= m_lowerCalPoint.yValue, 
															maxOutput	:= m_upperCalPoint.yValue),
								maxFlow	:= m_flowMax);
	END_IF
	
	m_upperCalTrigger(CLK:= (NOT m_pTransducer^.IsZeroCalRunning()) AND (m_calibrateHighPoint));
	IF (m_upperCalTrigger.Q) THEN
		m_upperCalPoint.xValue	:= m_pTransducer^.GetZeroCalValue();
		
		m_calibrateHighPoint := FALSE;
		
		// Calculate a new maximum flow
		SetFlowRange_MinMax(	minFlow := m_flowMin,
								maxFlow	:= f_LinearScale(	value		:= m_pTransducer^.GetMaxOutput(), 
															minInput	:= m_lowerCalPoint.xValue, 
															maxInput	:= m_upperCalPoint.xValue, 
															minOutput	:= m_lowerCalPoint.yValue, 
															maxOutput	:= m_upperCalPoint.yValue));
	END_IF
	
	// Set the raw flow value in the base flow meter class in volume/t units
	//SetRawFlow(flow:= f_LinearScale(	value		:= m_pTransducer^.signalValue, 
	//									minInput	:= m_pTransducer^.GetMinOutput(), 
	//									maxInput	:= m_pTransducer^.GetMaxOutput(), 
	//									minOutput	:= m_flowMin, 
	//									maxOutput	:= m_flowMax);
	IF (NOT m_pTransducer^.IsZeroCalRunning()) THEN
		SetRawFlow(flow:= f_LinearScale(	value		:= m_pTransducer^.signalValue, 
											minInput	:= m_lowerCalPoint.xValue, 
											maxInput	:= m_upperCalPoint.xValue, 
											minOutput	:= m_lowerCalPoint.yValue, 
											maxOutput	:= m_upperCalPoint.yValue));
	END_IF
								
ELSE

	SetRawFlow(flow:= 0.0);

END_IF
						
// Output the corrected Flow Value in voume/t units
correctedFlow := GetCorrectedFlow();

// Update the totalizers in voume/t units
m_totalizer1(	inputRate	:= MAX(0, GetCorrectedFlow()), 
				totalValue	=> m_total1);
				
m_totalizer2(	inputRate	:= MAX(0, GetCorrectedFlow()), 
				totalValue	=> m_total2);
				
m_totalizer3(	inputRate	:= MAX(0, GetCorrectedFlow()), 
				totalValue	=> m_total3);
				
// Update Alarms
m_LowFlowLimitAlarm.MonitorReal(	value	:= correctedFlow);
m_LowFlowWarningAlarm.MonitorReal(	value	:= correctedFlow);
m_HighFlowWarningAlarm.MonitorReal(	value	:= correctedFlow);
m_HighFlowLimitAlarm.MonitorReal(	value	:= correctedFlow);

(* ---------------------------------------------------------------------------
Func name   : 	CalibrateHighDataPoint
Description : 	Averages the transducer signal input value to provide
				a high calibration data point for the flowmeter scale.
Inputs      :	val			-	Calibration value in volume/t units
				duration_ms	-	Duration of value averaging time in ms
Returns     : 	None
Notes       : 	
--------------------------------------------------------------------------- *)

METHOD CalibrateHighDataPoint
VAR_INPUT
	val				: REAL;		// Calibration value in volume/t units
	duration_ms 	: UINT;		// Duration of value averaging time in ms
END_VAR
IF ((NOT m_calibrateLowPoint) AND (NOT m_calibrateHighPoint)) THEN
	m_pTransducer^.ZeroCal(duration_ms:= duration_ms);
	m_upperCalPoint.yValue	:= val;
	m_calibrateHighPoint := TRUE;
END_IF
END_METHOD

(* ---------------------------------------------------------------------------
Func name   : 	CalibrateLowDataPoint
Description : 	Averages the transducer signal input value to provide
				a low calibration data point for the flowmeter scale.
Inputs      :	val			-	Calibration value in volume/t units
				duration_ms	-	Duration of value averaging time in ms
Returns     : 	None
Notes       : 	
--------------------------------------------------------------------------- *)

METHOD CalibrateLowDataPoint
VAR_INPUT
	val				: REAL;		// Calibration value in volume/t units
	duration_ms 	: UINT;		// Duration of value averaging time in ms
END_VAR
VAR
	minFlow		: REAL;
	maxFlow		: REAL;
END_VAR
IF ((NOT m_calibrateLowPoint) AND (NOT m_calibrateHighPoint)) THEN
	m_pTransducer^.ZeroCal(duration_ms:= duration_ms);
	m_lowerCalPoint.yValue	:= val;
	m_calibrateLowPoint := TRUE;
END_IF
END_METHOD

(* ---------------------------------------------------------------------------
Func name   : 	ClearCalibration
Description : 	Clears all calibration of the flowmeter and resets to
				the default constructor scale.
Inputs      :	None
Returns     : 	None
Notes       : 	
--------------------------------------------------------------------------- *)

METHOD ClearCalibration
VAR_INPUT
END_VAR
// Reset to default values
m_lowerCalPoint.xValue	:= m_pTransducer^.GetMinOutput();
m_lowerCalPoint.yValue	:= m_defaultFlowMin;

m_upperCalPoint.xValue	:= m_pTransducer^.GetMaxOutput();
m_upperCalPoint.yValue	:= m_defaultFlowMax;

SetFlowRange_MinMax(	minFlow := m_defaultFlowMin,
						maxFlow	:= m_defaultFlowMax);
						
m_calibrateLowPoint		:= FALSE;
m_calibrateHighPoint	:= FALSE;
END_METHOD

(* ---------------------------------------------------------------------------
Func name   : 	FB_exit
Description : 	Destructor
Inputs      :	None
Returns     : 	None
Notes       : 	
--------------------------------------------------------------------------- *)

METHOD FB_exit : BOOL
VAR_INPUT
	bInCopyCode : BOOL; // if TRUE, the exit method is called for exiting an instance that is copied afterwards (online change)
END_VAR
// Do nothing
END_METHOD

(* ---------------------------------------------------------------------------
Func name   : 	FB_init
Description : 	Constructor
Inputs      :	pTransducer			:	transducer pointer
				minFlow				: 	minimum flow value at transducer minimum value (volume/t)
				maxFlow				:	maximum flow value at transducer maximum value (volume/t)
Returns     : 	None
Notes       : 	
--------------------------------------------------------------------------- *)

METHOD FB_init : BOOL
VAR_INPUT
	bInitRetains 		: BOOL; 							// if TRUE, the retain variables are initialized (warm start / cold start)
    bInCopyCode  		: BOOL; 							// if TRUE, the instance afterwards gets moved into the copy code (online change)
	pTransducer 		: POINTER TO fb_AnalogTransducer;	// transducer pointer
	minFlow 			: REAL;								// minimum flow value at transducer minimum value (volume/t)
	maxFlow 			: REAL;								// maximum flow value at transducer maximum value (volume/t)
END_VAR
// Default User kFact to 1.0
SetUserKFact(kfact := 1.0);

// Default the raw flow value to 0
SetRawFlow(flow:= 0.0);

// Initialize / Reset the totalizers
m_totalizer1.Reset();
m_totalizer2.Reset();
m_totalizer1.Reset();

// Enable the totalizers as default
m_totalizer1.Enable();
m_totalizer2.Enable();
m_totalizer3.Enable();

// Set the flow ranges in volume/t units
m_defaultFlowMin		:= minFlow;				// in volume/t units
m_defaultFlowMax 		:= maxFlow;				// in volume/t units
SetFlowRange_MinMax(	minFlow := minFlow,
						maxFlow	:= maxFlow);
						
// Set the transducer pointer
m_pTransducer := pTransducer;

// Initialize the calibration values
m_lowerCalPoint.xValue	:= m_pTransducer^.GetMinOutput();
m_lowerCalPoint.yValue	:= minFlow;

m_upperCalPoint.xValue	:= m_pTransducer^.GetMaxOutput();
m_upperCalPoint.yValue	:= maxFlow;


m_lowerCalTrigger(CLK:= FALSE);
m_upperCalTrigger(CLK:= FALSE);
m_calibrateLowPoint		:= FALSE;
m_calibrateHighPoint	:= FALSE;
END_METHOD

(* ---------------------------------------------------------------------------
Func name   : 	GetLowerCalDataPoint
Description : 	returns the flowmeter lower calibration data point.
Inputs      :	None
Returns     : 	REAL	-	lower calibration data point
Notes       : 	
--------------------------------------------------------------------------- *)

METHOD GetLowerCalDataPoint : TCalibrationDataPoint
VAR_INPUT
END_VAR
GetLowerCalDataPoint := m_lowerCalPoint;
END_METHOD

(* ---------------------------------------------------------------------------
Func name   : 	GetUpperCalDataPoint
Description : 	returns the flowmeter upper calibration data point.
Inputs      :	None
Returns     : 	REAL	-	upper calibration data point
Notes       : 	
--------------------------------------------------------------------------- *)

METHOD GetUpperCalDataPoint : TCalibrationDataPoint
VAR_INPUT
END_VAR
GetUpperCalDataPoint := m_upperCalPoint;
END_METHOD

(* ---------------------------------------------------------------------------
Func name   : 	SetLowerCalDataPoint
Description : 	sets the flowmeter lower calibration data point.
Inputs      :	calPoint	-	calibration data point
Returns     : 	None
Notes       : 	
--------------------------------------------------------------------------- *)

METHOD SetLowerCalDataPoint
VAR_INPUT
	calPoint	: TCalibrationDataPoint;
END_VAR
m_lowerCalPoint := calPoint;
END_METHOD

(* ---------------------------------------------------------------------------
Func name   : 	SetUpperCalDataPoint
Description : 	sets the flowmeter upper calibration data point.
Inputs      :	calPoint	-	calibration data point
Returns     : 	None
Notes       : 	
--------------------------------------------------------------------------- *)

METHOD SetUpperCalDataPoint
VAR_INPUT
	calPoint	: TCalibrationDataPoint;
END_VAR
m_upperCalPoint := calPoint;
END_METHOD

END_FUNCTION_BLOCK

// 20 Program Organization Units/Instrument-Controller Functions/fb_FlowMeter
(*AUTHOR:			Jaison Schaab*)
(*DATE:				June 9 / 2020*)
(*DESCRIPTION: 		This Function Block provides a BASE class for all flow meter objects.  The class
					consists of the following features:
					
						-	Min/Max configurable flow ranges in volume/t units whose range/values define the flow units of the entire class
						-	Raw volume flow value in volume/t units which is to be set by the derived class from its data source
						-	User settable unitless k-factor value which allows corrections in the flow value
						-	Corrected volume flow value in volume/t units which is the raw flow with k-factor applied
						-	Automatic k-factor calculation given known reference flow in volume/t units
						-	3 seperate volume flow totalizers with pause/resume/reset functionality
					
					No Alarms are currently included. however alarm handler / fault function are defined.*)

(*UPDATE: 			March. 23 2021 - Jaison Schaab

					Code Is fully tested and functional.				
*)

(*UPDATE: 			March. 18 2021 - Jaison Schaab

					Code Ported from Wago.
					
					Code has NOT Yet been tested.
*)

(*UPDATE: 			August. 31 2020 - Jaison Schaab

					Added "m_defaultFlowMin" and "m_defaultFlowMax" values which will allow the flow meter range
					to be re-defined through calibration and then restored to orginal constructor limits.
*)	

(*UPDATE: 			June. 23 2020 - Jaison Schaab

					Removed backdoor (m_pAlarmHandler : POINTER TO fb_AlarmHandler) alarm handler function pointer
					in order to simplify the alarm system.  Any alarms at this level should define a instance
					of the fb_AlarmMonitor class which will handle the alarm registration/set/clear.
*)	

(*NOTES:			The derived flow meter class is required to:
					
						- 	Define and set the m_flowMin/m_flowMax values in the desired volume flow units.
							For example if the range of (0 - 10 m3/min) then all values in that flowmeter instance
							 will return values in m3/min.  Including raw/corrected flow and all totalizers.
						-	Set the m_rawFlow value in volume/t units using the SetRawFlow() method.
						-	cyclically call the 3 totalizer objects to ensure they are updated on each scan.
						-	Initialize all values in the constructor including the user k-factor, totalizer
							reset/enable, and setting the alarm handler pointer.

*)

FUNCTION_BLOCK fb_FlowMeter
VAR_INPUT
END_VAR
VAR_OUTPUT
END_VAR
VAR
	// Default constructor flow limits
	m_defaultFlowMin		: REAL			:= 0.0;			// in volume/t units
	m_defaultFlowMax 		: REAL			:= 0.0;			// in volume/t units	
	
	// Current configured flow limits
	m_flowMin				: REAL			:= 0.0;			// in volume/t units
	m_flowMax 				: REAL			:= 0.0;			// in volume/t units	

	m_rawFlow				: REAL			:= 0.0;			// in volume/t units

	// Config Variables
	m_userkfact				: REAL			:= 1.0;			// unitless multiplier (1.0 simply allows raw value output)
	
	m_total1				: REAL			:= 0.0;			// in volume/t units
	m_total2				: REAL			:= 0.0;			// in volume/t units
	m_total3				: REAL			:= 0.0;			// in volume/t units
	
	m_totalizer1			: Totalizer;					// totalizer 1
	m_totalizer2			: Totalizer;					// totalizer 2
	m_totalizer3			: Totalizer;					// totalizer 3
	
	// Fault Handling (Alarms)
	m_devId					: UDeviceId;					// Device Id used for alarm integration
	
	// Alarms
	m_LowFlowLimitAlarm 	: fb_AlarmMonitor;				// Alarm - Low flow limit alarm
	m_LowFlowWarningAlarm 	: fb_AlarmMonitor;				// Alarm - Low flow warning alarm
	m_HighFlowWarningAlarm 	: fb_AlarmMonitor;				// Alarm - high flow warning alarm
	m_HighFlowLimitAlarm 	: fb_AlarmMonitor;				// Alarm - high flow limit alarm
	
END_VAR
VAR CONSTANT
	USER_K_FACTOR_MIN		: REAL := 0.1;					// minimum allowable user k-factor
	USER_K_FACTOR_MAX		: REAL := 10.0;					// maximum allowable user k-factor
	ALARM_HYST_PERCENT		: REAL := 1.0;					// hysteresis percentage for reseting alarms
END_VAR

(* ---------------------------------------------------------------------------
Func name   : 	CalculateUserKFact
Description : 	Routine will calculate and set the flow meter k-factor
				so that the corrected flow matches the input reference
				flow value.
Inputs      :	refFlow	-	reference flow value in volume/t
Returns     : 	None
Notes       : 	Use this routine to calibrate the flow meter to a known
				flow in volume/t.
--------------------------------------------------------------------------- *)

METHOD CalculateUserKFact
VAR_INPUT
	refFlow	: REAL;
END_VAR
IF (m_rawFlow > 0.0) THEN
	SetUserKFact(refFlow / m_rawFlow);
END_IF
END_METHOD

(* ---------------------------------------------------------------------------
Func name   : 	GetCorrectedFlow
Description : 	Routine to calculate and return the corrected volume flow
				with the user k-factor applied in volume/t units.
Inputs      :	None
Returns     : 	REAL	-	The corrected volume flow value in volume/t
Notes       : 	
--------------------------------------------------------------------------- *)

METHOD GetCorrectedFlow : REAL
VAR_INPUT
END_VAR
GetCorrectedFlow := m_userkfact * m_rawFlow;
END_METHOD

(* ---------------------------------------------------------------------------
Func name   : 	GetFlowRange_MinMax
Description : 	Gets the minimum/maximum flow range values from the flowmeter
				in volume/t units.
Inputs      :	None
Returns     : 	minFlow		: 	flowmeter minimum flow value (volume/t)
				maxFlow		:	flowmeter maximum flow value (volume/t)
Notes       : 	
--------------------------------------------------------------------------- *)

METHOD GetFlowRange_MinMax
VAR_INPUT
END_VAR
VAR_OUTPUT
	minFlow 	: REAL;		// minimum flow value at transducer minimum value (volume/t)
	maxFlow 	: REAL;		// maximum flow value at transducer maximum value (volume/t)
END_VAR
// output the min/max flowmeter ranges
minFlow := m_flowMin;
maxFlow := m_flowMax;
END_METHOD

(* ---------------------------------------------------------------------------
Func name   : 	GetRawFlow
Description : 	Routine to return the raw volume flow value in volume/t units.
				This value does not have the k-factor applied.
Inputs      :	None
Returns     : 	REAL	-	The raw volume flow value in volume/t
Notes       : 	
--------------------------------------------------------------------------- *)

METHOD GetRawFlow : REAL
VAR_INPUT
END_VAR
GetRawFlow := m_rawFlow;
END_METHOD

(* ---------------------------------------------------------------------------
Func name   : 	GetUserAlarms
Description : 	Gets the low/high flow warning alarm value in volume/t units.
Inputs      :	None
Returns     : 	lowFlowWarn		: 	low flow warning alarm value (volume/t)
				highFlowWarn	:	high flow warning alarm value (volume/t)
Notes       : 	
--------------------------------------------------------------------------- *)

METHOD GetUserAlarms
VAR_INPUT
END_VAR
VAR_OUTPUT
	lowFlowWarn 	: REAL;		// low flow warning alarm value (volume/t)
	highFlowWarn	: REAL;		// high flow warning alarm value (volume/t)
END_VAR
lowFlowWarn  	:= LREAL_TO_REAL(m_LowFlowWarningAlarm.m_limit.limitOn);
highFlowWarn  	:= LREAL_TO_REAL(m_HighFlowWarningAlarm.m_limit.limitOn);
END_METHOD

(* ---------------------------------------------------------------------------
Func name   : 	GetUserKFact
Description : 	Routine will return the unitless user k-factor value.
Inputs      :	None
Returns     : 	REAL	-	The unitless user k-factor value
Notes       : 	
--------------------------------------------------------------------------- *)

METHOD GetUserKFact : REAL
VAR_INPUT
END_VAR
GetUserKFact := m_userkfact;
END_METHOD

(* ---------------------------------------------------------------------------
Func name   : 	GetVolumeTotal1
Description : 	Routine to return the current volume totalizer 1 value 
				in volume/t units.
Inputs      :	None
Returns     : 	REAL	-	Totalizer 1 volume flow value in volume/t
Notes       : 	
--------------------------------------------------------------------------- *)

METHOD GetVolumeTotal1 : REAL
VAR_INPUT
END_VAR
GetVolumeTotal1 := m_total1;
END_METHOD

(* ---------------------------------------------------------------------------
Func name   : 	GetVolumeTotal2
Description : 	Routine to return the current volume totalizer 2 value 
				in volume/t units.
Inputs      :	None
Returns     : 	REAL	-	Totalizer 2 volume flow value in volume/t
Notes       : 	
--------------------------------------------------------------------------- *)

METHOD GetVolumeTotal2 : REAL
VAR_INPUT
END_VAR
GetVolumeTotal2 := m_total2;
END_METHOD

(* ---------------------------------------------------------------------------
Func name   : 	GetVolumeTotal3
Description : 	Routine to return the current volume totalizer 3 value 
				in volume/t units.
Inputs      :	None
Returns     : 	REAL	-	Totalizer 3 volume flow value in volume/t
Notes       : 	
--------------------------------------------------------------------------- *)

METHOD GetVolumeTotal3 : REAL
VAR_INPUT
END_VAR
GetVolumeTotal3 := m_total3;
END_METHOD

(* ---------------------------------------------------------------------------
Func name   : 	InitAlarms
Description : 	Initializes the deviceId member variable used to set/clear
				the approproate alarms.
Inputs      :	None
Returns     : 	None
Notes       : 	
--------------------------------------------------------------------------- *)

METHOD InitAlarms
VAR_INPUT
	devId		: UDeviceId;	// Device Id used for alarm integration
END_VAR
// Set the device id which is used for alarm integrtion
m_devId := devId;

// Initialize the low flow limit alarm - Set to m_flowMin
m_LowFlowLimitAlarm.InitAlarm(code:= f_AlarmCode(devId:= devId, code:= f_FaultCode(TFaultPriority.Error, TFaultCondition.UnderLimit)), alarmType:= TAlarmMonitorType.lower_limit, delayTime:= T#0S);
m_LowFlowLimitAlarm.SetLimitReal(on:= m_flowMin, off:= m_flowMin + MAX(0.001, (ABS(m_flowMin) * (ALARM_HYST_PERCENT / 100.0))));
m_LowFlowLimitAlarm.EnableLimit();
	
// Initialize the low flow warning alarm - Default to disabled
m_LowFlowWarningAlarm.InitAlarm(code:= f_AlarmCode(devId:= devId, code:= f_FaultCode(TFaultPriority.Warning, TFaultCondition.UnderWarning)), alarmType:= TAlarmMonitorType.lower_limit, delayTime:= T#0S);
m_LowFlowWarningAlarm.DisableLimit();

// Initialize the high flow warning alarm - Default to disabled
m_HighFlowWarningAlarm.InitAlarm(code:= f_AlarmCode(devId:= devId, code:= f_FaultCode(TFaultPriority.Warning, TFaultCondition.OverWarning)), alarmType:= TAlarmMonitorType.upper_limit, delayTime:= T#0S);
m_HighFlowWarningAlarm.DisableLimit();

// Initialize the high flow limit alarm - Set to m_flowMax
m_HighFlowLimitAlarm.InitAlarm(code:= f_AlarmCode(devId:= devId, code:= f_FaultCode(TFaultPriority.Error, TFaultCondition.OverLimit)), alarmType:= TAlarmMonitorType.upper_limit, delayTime:= T#0S);
m_HighFlowLimitAlarm.SetLimitReal(on:= m_flowMax, off:= m_flowMax - MAX(0.001, (ABS(m_flowMax) * (ALARM_HYST_PERCENT / 100.0))));
m_HighFlowLimitAlarm.EnableLimit();
END_METHOD

(* ---------------------------------------------------------------------------
Func name   : 	PauseVolumeTotal1
Description : 	Routine to pause volume totalizer 1.
Inputs      :	None
Returns     : 	None
Notes       : 	
--------------------------------------------------------------------------- *)

METHOD PauseVolumeTotal1
VAR_INPUT
END_VAR
m_totalizer1.Disable();
END_METHOD

(* ---------------------------------------------------------------------------
Func name   : 	PauseVolumeTotal2
Description : 	Routine to pause volume totalizer 2.
Inputs      :	None
Returns     : 	None
Notes       : 	
--------------------------------------------------------------------------- *)

METHOD PauseVolumeTotal2
VAR_INPUT
END_VAR
m_totalizer2.Disable();
END_METHOD

(* ---------------------------------------------------------------------------
Func name   : 	PauseVolumeTotal3
Description : 	Routine to pause volume totalizer 3.
Inputs      :	None
Returns     : 	None
Notes       : 	
--------------------------------------------------------------------------- *)

METHOD PauseVolumeTotal3
VAR_INPUT
END_VAR
m_totalizer3.Disable();
END_METHOD

(* ---------------------------------------------------------------------------
Func name   : 	ResetVolumeTotal1
Description : 	Routine to reset volume totalizer 1 to 0.
Inputs      :	None
Returns     : 	None
Notes       : 	
--------------------------------------------------------------------------- *)

METHOD ResetVolumeTotal1
VAR_INPUT
END_VAR
m_totalizer1.Reset();
m_total1 := 0.0;
END_METHOD

(* ---------------------------------------------------------------------------
Func name   : 	ResetVolumeTotal2
Description : 	Routine to reset volume totalizer 2 to 0.
Inputs      :	None
Returns     : 	None
Notes       : 	
--------------------------------------------------------------------------- *)

METHOD ResetVolumeTotal2
VAR_INPUT
END_VAR
m_totalizer2.Reset();
m_total2 := 0.0;
END_METHOD

(* ---------------------------------------------------------------------------
Func name   : 	ResetVolumeTotal3
Description : 	Routine to reset volume totalizer 3 to 0.
Inputs      :	None
Returns     : 	None
Notes       : 	
--------------------------------------------------------------------------- *)

METHOD ResetVolumeTotal3
VAR_INPUT
END_VAR
m_totalizer3.Reset();
m_total3 := 0.0;
END_METHOD

(* ---------------------------------------------------------------------------
Func name   : 	ResumeVolumeTotal1
Description : 	Routine to resume volume totalizer 1.
Inputs      :	None
Returns     : 	None
Notes       : 	
--------------------------------------------------------------------------- *)

METHOD ResumeVolumeTotal1
VAR_INPUT
END_VAR
m_totalizer1.Enable();
END_METHOD

(* ---------------------------------------------------------------------------
Func name   : 	ResumeVolumeTotal2
Description : 	Routine to resume volume totalizer 2.
Inputs      :	None
Returns     : 	None
Notes       : 	
--------------------------------------------------------------------------- *)

METHOD ResumeVolumeTotal2
VAR_INPUT
END_VAR
m_totalizer2.Enable();
END_METHOD

(* ---------------------------------------------------------------------------
Func name   : 	ResumeVolumeTotal3
Description : 	Routine to resume volume totalizer 3.
Inputs      :	None
Returns     : 	None
Notes       : 	
--------------------------------------------------------------------------- *)

METHOD ResumeVolumeTotal3
VAR_INPUT
END_VAR
m_totalizer3.Enable();
END_METHOD

(* ---------------------------------------------------------------------------
Func name   : 	SetFlowRange_MinMax
Description : 	Sets the minimum/maximum flow range values for the flowmeter
				in volume/t units.  The units defined by this range will
				define the units for all flow meter values.
Inputs      :	minFlow		: 	flowmeter minimum flow value (volume/t)
				maxFlow		:	flowmeter maximum flow value (volume/t)
Returns     : 	TRUE on success, else FALSE
Notes       : 	For example if the range of (0 - 10 m3/min) then all values 
				in that flowmeter instance should be interpreted as m3/min.  
				Including raw/corrected flow and all totalizers.
--------------------------------------------------------------------------- *)

METHOD SetFlowRange_MinMax : BOOL
VAR_INPUT
	minFlow 	: REAL;		// minimum flow value at transducer minimum value (volume/t)
	maxFlow 	: REAL;		// maximum flow value at transducer maximum value (volume/t)
END_VAR
// Check to ensure max is larger than min
IF (maxFlow > minFlow) THEN
	
	// Set the min/max flowmeter ranges
	m_flowMin := minFlow;
	m_flowMax := maxFlow;
	
	SetFlowRange_MinMax := TRUE;
	
	// Configure / Enable the low flow limit alarm
	m_LowFlowLimitAlarm.SetLimitReal(on:= m_flowMin, off:= m_flowMin + MAX(0.001, (ABS(m_flowMin) * (ALARM_HYST_PERCENT / 100.0))));
	m_LowFlowLimitAlarm.EnableLimit();
	
	// Configure / Enable the high flow limit alarm
	m_HighFlowLimitAlarm.SetLimitReal(on:= m_flowMax, off:= m_flowMax - MAX(0.001, (ABS(m_flowMax) * (ALARM_HYST_PERCENT / 100.0))));
	m_HighFlowLimitAlarm.EnableLimit();
	
ELSE
	
	SetFlowRange_MinMax := FALSE;

END_IF
END_METHOD

(* ---------------------------------------------------------------------------
Func name   : 	SetFlow
Description : 	Priavte function which allows the derived classes to sets the 
				flowmeter rawFlow value in volume/t units.  
Inputs      :	flow	-	raw flow rate in volume/t units
Returns     : 	REAL	-	actual set raw flow rate in volume/t units
Notes       : 	The value will be limited by the initialized 
				minFlow/maxFlow values.
--------------------------------------------------------------------------- *)

METHOD PROTECTED SetRawFlow : REAL
VAR_INPUT
	flow	: REAL;		// in volume/t units
END_VAR
// Set the raw flow value in the base flow meter class in volume/t units
m_rawFlow := MAX(MIN(flow, m_flowMax), m_flowMin);

// Return actual set flow
SetRawFlow := m_rawFlow;
END_METHOD

(* ---------------------------------------------------------------------------
Func name   : 	SetUserAlarms
Description : 	Sets the low/high flow warning alarm values in volume/t units.
Inputs      :	lowFlowWarn		: 	low flow warning alarm value (volume/t)
				highFlowWarn	:	high flow warning alarm value (volume/t)
Returns     : 	TRUE on success, else FALSE
Notes       : 	The values will be checked against the configured min/max flow
				range of the meter and capped at those values.  A hysteresis
				will be applied for the reset value. If the high flow value is
				not greater than the low flow value nothing will happen.
--------------------------------------------------------------------------- *)

METHOD SetUserAlarms : BOOL
VAR_INPUT
	lowFlowWarn 	: REAL;		// low flow warning alarm value (volume/t)
	highFlowWarn	: REAL;		// high flow warning alarm value (volume/t)
END_VAR
// Configure / Enable the low flow warning alarm
IF ((lowFlowWarn = NOTUSED) OR (lowFlowWarn <= m_flowMin)) THEN
	lowFlowWarn := m_flowMin;
	m_LowFlowWarningAlarm.DisableLimit();
ELSE
	m_LowFlowWarningAlarm.EnableLimit();
END_IF

m_LowFlowWarningAlarm.SetLimitReal(on:= lowFlowWarn, off:= lowFlowWarn + MAX(0.001, (ABS(lowFlowWarn) * (ALARM_HYST_PERCENT / 100.0))));
		
// Configure / Enable the high flow warning alarm
IF ((highFlowWarn = NOTUSED) OR (highFlowWarn > m_flowMax)) THEN
	highFlowWarn := m_flowMax;
	m_HighFlowWarningAlarm.DisableLimit();
ELSE
	m_HighFlowWarningAlarm.EnableLimit();
END_IF

m_HighFlowWarningAlarm.SetLimitReal(on:= highFlowWarn, off:= highFlowWarn - MAX(0.001, (ABS(highFlowWarn) * (ALARM_HYST_PERCENT / 100.0))));
	
SetUserAlarms := TRUE;
END_METHOD

(* ---------------------------------------------------------------------------
Func name   : 	SetUserKFact
Description : 	Routine to set the unitless user k-factor value.
Inputs      :	kfact	-	The desried unitless user k-factor value
Returns     : 	None
Notes       : 	The value will be limited by the constants 
				USER_K_FACTOR_MIN and USER_K_FACTOR_MAX.
--------------------------------------------------------------------------- *)

METHOD SetUserKFact
VAR_INPUT
	kfact	: REAL;
END_VAR
m_userkfact := MAX(MIN(kfact, USER_K_FACTOR_MAX), USER_K_FACTOR_MIN);
END_METHOD

END_FUNCTION_BLOCK

// 20 Program Organization Units/Utility Functions/Totalizer
(*UPDATE: 			March. 23 2021 - Jaison Schaab

					Code Is fully tested and functional.				
*)

(*UPDATE: 			March. 18 2021 - Jaison Schaab

					Code Ported from Wago.
					
					Code has NOT Yet been tested.
*)

FUNCTION_BLOCK Totalizer
VAR_INPUT
	/// Units/min
	inputRate: REAL;
END_VAR
VAR_OUTPUT
	/// Total value in Units
	totalValue: REAL;
END_VAR
VAR
	isDisabled: BOOL;
	timeDifference: REAL;
	lastCallTime: DWORD;
	/// Saved integer portion of the total value
	integerTotal: UDINT;
	/// Saved decimal portion of the total value
	decimalTotal: REAL;
	/// currentStep is the change in the total that will be applied based on the input rate and time difference.
	currentStep: REAL;
	integerStep: UDINT;
END_VAR
VAR CONSTANT
	MIN_TO_MS: REAL := 1.67E-05;
END_VAR

// When the block is disabled, no changes should be recorded.
IF isDisabled THEN
	// Keep the call time up-to-date to avoid a large step upon falling edge of isDisabled.
	lastCallTime := SysTimeGetMs();
	RETURN;
END_IF

// Calculate the difference in time between the previous and current cycles
timeDifference := DWORD_TO_REAL( SysTimeGetMs() - lastCallTime );

// Calculate the current step in units/ms
currentStep := decimalTotal + inputRate * MIN_TO_MS * timeDifference;

// Isolate the integer portion of the current step
integerStep := TO_UDINT( TRUNC( currentStep ) );

// Increment stored portions of the total value
integerTotal := integerTotal + integerStep;
decimalTotal := currentStep - TO_REAL(integerStep);

// Sum the stored total into single output value
totalValue := decimalTotal + TO_REAL(integerTotal);

// Save current system time for use in next cycle
lastCallTime := SysTimeGetMs();

METHOD Disable : BOOL
isDisabled := TRUE;

// Returns TRUE to show the method was run
Disable := TRUE;
END_METHOD

METHOD Enable : BOOL
isDisabled := FALSE;

// Returns TRUE to show the method was run
Enable := TRUE;
END_METHOD

METHOD FB_Init : BOOL
VAR_INPUT
	/// if TRUE, the retain variables are initialized (warm start / cold start)
	bInitRetains: BOOL;
	/// if TRUE, the instance afterwards gets moved into the copy code (online change)
	bInCopyCode: BOOL;
END_VAR
// Initialize lastCallTime to be the current system time so the initial total starts at zero
lastCallTime := SysTimeGetMs();
END_METHOD

METHOD Reset : BOOL
decimalTotal := 0;
integerTotal := 0;
totalValue := 0;
END_METHOD

METHOD SetTotal : BOOL
VAR_INPUT
	/// Value to be set as new total
	setValue: REAL;
END_VAR
// Split total value into integer and franctional portions to maintain precision 
integerTotal := TO_UDINT( TRUNC( setValue ) );
decimalTotal := setValue - TO_REAL( TRUNC( setValue ) );

totalValue := UDINT_TO_REAL( integerTotal ) + decimalTotal;

// Returns TRUE to show the method was run
SetTotal := TRUE;
END_METHOD

END_FUNCTION_BLOCK

// 20 Program Organization Units/Instrument-Controller Functions/fb_ENDP_Freq_Tachometer
(*UPDATE: 			March. 18 2021 - Jaison Schaab

					Code Ported from Wago.
					
					Code has NOT Yet been tested.
*)

(*UPDATE: 			June. 23 2020 - Jaison Schaab

					Removed backdoor (m_pAlarmHandler : POINTER TO fb_AlarmHandler) alarm handler function pointer
					in order to simplify the alarm system.  Any alarms at this level should define a instance
					of the fb_AlarmMonitor class which will handle the alarm registration/set/clear.
*)	

FUNCTION_BLOCK fb_ENDP_Freq_Tachometer
VAR_INPUT
	//input_hz : REAL; use P_TO txducer to get value in Hz. It will be already filtered thru HistAvg(10,2)
END_VAR
VAR_OUTPUT
	output_rpm : REAL;
	endpState : INT;
END_VAR
VAR
	m_pFreqTransducer : POINTER TO fb_FreqTransducer;
	m_ppr : REAL;
END_VAR

output_rpm := REAL_TO_INT( m_pFreqTransducer^.freqValue * 60.0 / m_ppr );
IF (m_pFreqTransducer^.rawValue < 0) THEN
	endpState := TEnuHmiGaugeState.LowAlarm;
ELSE
	endpState := TEnuHmiGaugeState.No_Alarm;
END_IF

(* ---------------------------------------------------------------------------
Func name   : 	FB_init
Description : 	ENDP_Freq_Tachometer (calculates RPM off of Freq-mode card)
Inputs      :	ppr for the physical FreqTransducer sensor (see the project PDFs),
                pointer to fb_Txducer reading the freq.card inputs
Returns     : 	None
--------------------------------------------------------------------------- *)

METHOD FB_init : BOOL
VAR_INPUT
	bInitRetains 		: BOOL; 		// if TRUE, the retain variables are initialized (warm start / cold start)
    bInCopyCode  		: BOOL; 		// if TRUE, the instance afterwards gets moved into the copy code (online change)
	arg_cardreader : POINTER TO fb_FreqTransducer;
	arg_ppr : UINT;
END_VAR
m_pFreqTransducer := arg_cardreader;
m_ppr := arg_ppr;
END_METHOD

END_FUNCTION_BLOCK

// 20 Program Organization Units/Instrument-Controller Functions/fb_ENDP_FreqFlowmeter
(*AUTHOR:			Jaison Schaab*)
(*DATE:				July 15 / 2020*)
(*DESCRIPTION: 		Derived flow meter class which provides a frequency flow meter object.  The raw volume flow
					value is calculated from the configured "Frequency Transducer" object and configured
					PPR/kfact/timebase settings in volume/t units.*)				 				 

(*UPDATE: 			March. 18 2021 - Jaison Schaab

					Code Ported from Wago.
					
					Code has NOT Yet been tested.
*)

FUNCTION_BLOCK fb_ENDP_FreqFlowmeter EXTENDS fb_FlowMeter
VAR_INPUT
END_VAR
VAR_OUTPUT
	correctedFlow		: REAL;							// Corrected flow in volume/t units
END_VAR
VAR
// Transducer input
	m_pTransducer		: POINTER TO fb_FreqTransducer;	// Pointer to transducer

// Flowmeter settings
	m_PPR				: REAL;							// transducer pulses/rev
	m_kfact				: REAL;							// transducer volume/rev
	m_timebaseSeconds	: UINT;							// timebase in seconds (1 = volume/s, 60 = volume/min)
END_VAR

// Ensure transducer pointer is not NULL
IF (m_pTransducer <> _NULL) THEN

	// Set the raw flow value in the base flow meter class in volume/t units
	SetRawFlow(flow:= m_pTransducer^.freqValue 	/ m_PPR								// divide frequency by PPR for rev/sec
												* m_kfact							// multiply by kfact for volume/sec
												* UINT_TO_REAL(m_timebaseSeconds));	// multiply by timebase seconds for volume/timebase
												
ELSE

	SetRawFlow(flow:= 0.0);

END_IF
							
// Output the corrected Flow Value in voume/t units
correctedFlow := GetCorrectedFlow();

// Update the totalizers in voume/t units
m_totalizer1(	inputRate	:= GetCorrectedFlow(), 
				totalValue	=> m_total1);
				
m_totalizer2(	inputRate	:= GetCorrectedFlow(), 
				totalValue	=> m_total2);
				
m_totalizer3(	inputRate	:= GetCorrectedFlow(), 
				totalValue	=> m_total3);
				
// Update Alarms
m_LowFlowLimitAlarm.MonitorReal(	value	:= correctedFlow);
m_LowFlowWarningAlarm.MonitorReal(	value	:= correctedFlow);
m_HighFlowWarningAlarm.MonitorReal(	value	:= correctedFlow);
m_HighFlowLimitAlarm.MonitorReal(	value	:= correctedFlow);

(* ---------------------------------------------------------------------------
Func name   : 	FB_exit
Description : 	Destructor
Inputs      :	None
Returns     : 	None
Notes       : 	
--------------------------------------------------------------------------- *)

METHOD FB_exit : BOOL
VAR_INPUT
	bInCopyCode : BOOL; // if TRUE, the exit method is called for exiting an instance that is copied afterwards (online change)
END_VAR
// Do nothing
END_METHOD

(* ---------------------------------------------------------------------------
Func name   : 	FB_init
Description : 	Constructor
Inputs      :	pTransducer			:	transducer pointer
				minFlow				: 	minimum flow value at transducer minimum value (volume/t)
				maxFlow				:	maximum flow value at transducer maximum value (volume/t)
				PPR					: 	transducer pulses/rev
				kfact				:	transducer volume/rev
				timebaseSeconds		: 	timebase in seconds (1 = volume/s, 60 = volume/min, 3600 = volume/hour)
Returns     : 	None
Notes       : 	
--------------------------------------------------------------------------- *)

METHOD FB_init : BOOL
VAR_INPUT
	bInitRetains 		: BOOL; 							// if TRUE, the retain variables are initialized (warm start / cold start)
    bInCopyCode  		: BOOL; 							// if TRUE, the instance afterwards gets moved into the copy code (online change)
	pTransducer 		: POINTER TO fb_FreqTransducer;		// transducer pointer
	minFlow 			: REAL;								// minimum flow value at transducer minimum value (volume/t)
	maxFlow 			: REAL;								// maximum flow value at transducer maximum value (volume/t)
	PPR					: REAL;								// flowmeter PPR (pulses/rev)
	kfact				: REAL;								// flowmeter k-factor (volume/rev)
	timebaseSeconds		: UINT;								// timebase in seconds, (1s = volume/s, 60s = volume/min, 3600s = volume/hour)
END_VAR
// Default User kFact to 1.0
SetUserKFact(kfact := 1.0);

// Default the raw flow value to 0
SetRawFlow(flow:= 0.0);

// Initialize / Reset the totalizers
m_totalizer1.Reset();
m_totalizer2.Reset();
m_totalizer1.Reset();

// Enable the totalizers as default
m_totalizer1.Enable();
m_totalizer2.Enable();
m_totalizer3.Enable();

// Set the flow ranges in volume/t units
m_defaultFlowMin		:= minFlow;				// in volume/t units
m_defaultFlowMax 		:= maxFlow;				// in volume/t units
SetFlowRange_MinMax(	minFlow := minFlow,
						maxFlow	:= maxFlow);

// Set default flow meter settings
SetPPR(PPR);
SetKFact(kfact);
SetTimebase(timebaseSeconds);
						
// Set the transducer pointer
m_pTransducer := pTransducer;
END_METHOD

(* ---------------------------------------------------------------------------
Func name   : 	GetKFact
Description : 	Routine to get the flow meter k-factor value in volume/rev units.
Inputs      :	None
Returns     : 	REAL	-	The flow meter k-factor in volume/rev
Notes       : 	
--------------------------------------------------------------------------- *)

METHOD GetKFact : REAL
VAR_INPUT
END_VAR
GetKFact := m_kfact;
END_METHOD

(* ---------------------------------------------------------------------------
Func name   : 	GetPPR
Description : 	Routine to get the flow meter PPR in pulses/rev units.
Inputs      :	None
Returns     : 	REAL	-	The flow meter PPR in pulses/rev
Notes       : 	
--------------------------------------------------------------------------- *)

METHOD GetPPR : REAL
VAR_INPUT
END_VAR
GetPPR := m_PPR;
END_METHOD

(* ---------------------------------------------------------------------------
Func name   : 	GetTimebase
Description : 	Routine to get the flow meter timebase value in seconds.
Inputs      :	None
Returns     : 	REAL	-	The flow meter timebase in seconds
Notes       : 	1 = volume/s, 60 = volume/min, 3600 = volume/hour
--------------------------------------------------------------------------- *)

METHOD GetTimebase : UINT
VAR_INPUT
END_VAR
GetTimebase := m_timebaseSeconds;
END_METHOD

(* ---------------------------------------------------------------------------
Func name   : 	SetKFact
Description : 	Routine to set the flow meter k-factor value in volume/rev units.
Inputs      :	volumePerRev	-	The desired k-factor in volume/rev
Returns     : 	REAL			-	The set k-factor in volume/rev
Notes       : 	The value cannot be 0 and will be modified to ensure it is
				greater than 0.01.
--------------------------------------------------------------------------- *)

METHOD SetKFact : REAL
VAR_INPUT
	volumePerRev	: REAL;		// k-factor in volume/rev units
END_VAR
m_kfact := MAX(volumePerRev, 0.01);		// k-factor cannot be zero

SetKFact := m_kfact;
END_METHOD

(* ---------------------------------------------------------------------------
Func name   : 	SetPPR
Description : 	Routine to set the flow meter PPR value in pulses/rev units.
Inputs      :	pulsesPerRev	-	The desired PPR in pulses/rev
Returns     : 	REAL			-	The set PPR in pulses/rev
Notes       : 	The value cannot be 0 and will be modified to ensure it is
				greater than 0.01.
--------------------------------------------------------------------------- *)

METHOD SetPPR : REAL
VAR_INPUT
	pulsePerRev		: REAL;		// PPR in pulses/rev units
END_VAR
m_PPR := MAX(pulsePerREV, 0.01);		// PPR cannot be zero

SetPPR := m_PPR;
END_METHOD

(* ---------------------------------------------------------------------------
Func name   : 	SetTimebase
Description : 	Routine to get the flow meter timebase value in seconds.
Inputs      :	seconds	-	The desired timebase value in seconds
Returns     : 	UINT	-	The flow meter timebase in seconds
Notes       : 	1 = volume/s, 60 = volume/min, 3600 = volume/hour

				The value will be modified to ensure it is between
				1 second and 3600 seconds.
--------------------------------------------------------------------------- *)

METHOD SetTimebase : UINT
VAR_INPUT
	seconds		: UINT;		// timebase seconds
END_VAR
m_timebaseSeconds := MAX(1, MIN(seconds, 3600));	// Limit the time base to 1s = volume/s to 3600s = volume/hour

SetTimebase := m_timebaseSeconds;
END_METHOD

END_FUNCTION_BLOCK

// 20 Program Organization Units/Instrument-Controller Functions/fb_ENDP_SimulatedDensitometer
(*AUTHOR:			Ryan Herdian*)
(*DATE:				June 18, 2020*)
(*DESCRIPTION: 		Derived densitometer class which provides a simulated denso object.  The raw volume flow
					value is set by using the "SetSimDensity" routine in the configured density units.  The density value
					is assumed to be ideal and therefore the user k-factor is NOT settable (always 1.0).

					This class is intended as a testing tool to verify functionality which relies 
					on density to be present.*)

(*UPDATE: 			March. 18 2021 - Jaison Schaab

					Code Ported from Wago.
					
					Code has NOT Yet been tested.
*)

FUNCTION_BLOCK fb_ENDP_SimulatedDensitometer EXTENDS fb_Densitometer
VAR_INPUT
END_VAR
VAR_OUTPUT
	correctedDensity		: REAL;			// Corrected density in Specific Gravity Unit, [SGU]
END_VAR
VAR
END_VAR

// Output the corrected density in Specific Gravity Unit, [SGU]
correctedDensity	:= GetCorrectedDensitySGU();


// Ensure the simulated density value is ideal with the user k-factor always 1.0
IF (GetUserKFact() <> 1.0) THEN
	SetUserKFact(1.0);
END_IF

(* ---------------------------------------------------------------------------
Func name   : 	FB_exit
Description : 	Destructor
Inputs      :	None
Returns     : 	None
Notes       : 	
--------------------------------------------------------------------------- *)

METHOD FB_exit : BOOL
VAR_INPUT
	bInCopyCode : BOOL; // if TRUE, the exit method is called for exiting an instance that is copied afterwards (online change)
END_VAR
// Do Nothing
END_METHOD

(* ---------------------------------------------------------------------------
Func name   : 	FB_init
Description : 	Constructor
Inputs      :	minDensity			: 	minimum density value at transducer minimum value in density unit, e.g.: Specific Gravity Unit, [SGU]
				maxDensity			:	maximum density value at transducer maximum value in density unit, e.g.: Specific Gravity Unit, [SGU]
Returns     : 	None
Notes       : 	
--------------------------------------------------------------------------- *)

METHOD FB_init : BOOL
VAR_INPUT
	bInitRetains 		: BOOL; 							// if TRUE, the retain variables are initialized (warm start / cold start)
    bInCopyCode  		: BOOL; 							// if TRUE, the instance afterwards gets moved into the copy code (online change)
	minDensity 			: REAL;								// minimum Density value at transducer minimum value in density unit, e.g.: Specific Gravity Unit, [SGU]
	maxDensity 			: REAL;								// maximum Density value at transducer maximum value in density unit, e.g.: Specific Gravity Unit, [SGU]
END_VAR
// Default User kFact to 1.0
SetUserKFact(kfact := 1.0);

// Default the raw density value to 0
SetRawDensity(density:= 0.0);

// Set the density ranges in density unit, e.g.: Specific Gravity Unit, [SGU]
SetDensityRange_MinMax(	minDensity	:= minDensity, 
						maxDensity	:= maxDensity);
END_METHOD

(* ---------------------------------------------------------------------------
Func name   : 	SetSimDensity
Description : 	Sets the simulated density value in in density unit, e.g.: Specific Gravity Unit, [SGU].  
Inputs      :	density	-	desired simulated density in density unit, e.g.: Specific Gravity Unit, [SGU]
Returns     : 	None
Notes       : 	The value will be limited by the initialized 
				minDensity/maxDensity values.
--------------------------------------------------------------------------- *)

METHOD SetSimDensity
VAR_INPUT
	density		: REAL;		// in density unit, e.g.: Specific Gravity Unit, [SGU]
END_VAR
SetRawDensity(density:= density);
END_METHOD

END_FUNCTION_BLOCK

// 20 Program Organization Units/Instrument-Controller Functions/fb_ENDP_SimulatedFlowMeter
(*AUTHOR:			Jaison Schaab*)
(*DATE:				June 9 / 2020*)
(*DESCRIPTION: 		Derived flow meter class which provides a simulated flow meter object.  The raw volume flow
					value is set by using the "SetFlow" routine in the configured volume/t units.  The flow value
					is assumed to be ideal and therefore the user k-factor is NOT settable (always 1.0).

					This class is intended as a testing tool to verify functionality which relies 
					on flow to be present.*)

(*UPDATE: 			March. 23 2021 - Jaison Schaab

					Code Is fully tested and functional.				
*)

(*UPDATE: 			March. 18 2021 - Jaison Schaab

					Code Ported from Wago.
					
					Code has NOT Yet been tested.
*)

FUNCTION_BLOCK fb_ENDP_SimulatedFlowMeter EXTENDS fb_FlowMeter
VAR_INPUT
END_VAR
VAR_OUTPUT
	correctedFlow		: REAL;						// Corrected flow in volume/t units
END_VAR
VAR
			
END_VAR

// Output the corrected Flow Value in voume/t units
correctedFlow := GetCorrectedFlow();

// Update the totalizers in voume/t units
m_totalizer1(	inputRate	:= GetCorrectedFlow(), 
				totalValue	=> m_total1);
				
m_totalizer2(	inputRate	:= GetCorrectedFlow(), 
				totalValue	=> m_total2);
				
m_totalizer3(	inputRate	:= GetCorrectedFlow(), 
				totalValue	=> m_total3);

// Ensure the simulated flow value is ideal with the user k-factor always 1.0 <JAISON>			
IF (GetUserKFact() <> 1.0) THEN
	SetUserKFact(1.0);
END_IF

// Update Alarms
m_LowFlowLimitAlarm.MonitorReal(	value	:= correctedFlow);
m_LowFlowWarningAlarm.MonitorReal(	value	:= correctedFlow);
m_HighFlowWarningAlarm.MonitorReal(	value	:= correctedFlow);
m_HighFlowLimitAlarm.MonitorReal(	value	:= correctedFlow);

(* ---------------------------------------------------------------------------
Func name   : 	FB_exit
Description : 	Destructor
Inputs      :	None
Returns     : 	None
Notes       : 	
--------------------------------------------------------------------------- *)

METHOD FB_exit : BOOL
VAR_INPUT
	bInCopyCode : BOOL; // if TRUE, the exit method is called for exiting an instance that is copied afterwards (online change)
END_VAR
// Do nothing
END_METHOD

(* ---------------------------------------------------------------------------
Func name   : 	FB_init
Description : 	Constructor
Inputs      :	minFlow				: 	flowmeter minimum flow value (volume/t)
				maxFlow				:	flowmeter maximum flow value (volume/t)
Returns     : 	None
Notes       : 	
--------------------------------------------------------------------------- *)

METHOD FB_init : BOOL
VAR_INPUT
	bInitRetains 		: BOOL; 							// if TRUE, the retain variables are initialized (warm start / cold start)
    bInCopyCode  		: BOOL; 							// if TRUE, the instance afterwards gets moved into the copy code (online change)
	minFlow 			: REAL;								// minimum flow value at transducer minimum value (volume/t)
	maxFlow 			: REAL;								// maximum flow value at transducer maximum value (volume/t)
END_VAR
// Default User kFact to 1.0
SetUserKFact(kfact := 1.0);

// Default the raw flow value to 0
SetRawFlow(flow:= 0.0);

// Initialize / Reset the totalizers
m_totalizer1.Reset();
m_totalizer2.Reset();
m_totalizer1.Reset();

// Enable the totalizers as default
m_totalizer1.Enable();
m_totalizer2.Enable();
m_totalizer3.Enable();

// Set the flow ranges in volume/t units
m_defaultFlowMin		:= minFlow;				// in volume/t units
m_defaultFlowMax 		:= maxFlow;				// in volume/t units
SetFlowRange_MinMax(	minFlow := minFlow,
						maxFlow	:= maxFlow);
END_METHOD

(* ---------------------------------------------------------------------------
Func name   : 	SetSimFlow
Description : 	Sets the simulated flow value in volume/t units.  
Inputs      :	flow	-	desired simulated flow rate in volume/t units
Returns     : 	REAL	-	actual set simulated flow value in volume/t units
Notes       : 	The value will be limited by the initialized 
				minFlow/maxFlow values.
--------------------------------------------------------------------------- *)

METHOD SetSimFlow : REAL
VAR_INPUT
	flow	: REAL;		// in volume/t units
END_VAR
SetSimFlow := SetRawFlow(flow:= flow);
END_METHOD

END_FUNCTION_BLOCK

// 20 Program Organization Units/Instrument-Controller Functions/fb_Indicator
(*AUTHOR:			Jaison Schaab*)
(*DATE:				March 27 / 2020*)
(*DESCRIPTION: 		This Function Block provides a standard conrol interface for digital
					outputs of type BOOL.*)

(*NOTES:			
*)

(*UPDATE: 			March. 23 2021 - Jaison Schaab

					Code Is fully tested and functional.				
*)

(*UPDATE: 			March. 18 2021 - Jaison Schaab

					Code Ported from Wago.
					
					Code has NOT Yet been tested.
*)
						
FUNCTION_BLOCK fb_Indicator
VAR_INPUT
END_VAR
VAR_OUTPUT
END_VAR
VAR
	m_signal	: POINTER TO BOOL;	// Pointer to the output BOOL signal value
END_VAR

(* ---------------------------------------------------------------------------
Func name   : 	FB_exit
Description : 	Destructor
Inputs      :	None
Returns     : 	None
Notes       : 	
--------------------------------------------------------------------------- *)

METHOD FB_exit : BOOL
VAR_INPUT
	bInCopyCode : BOOL; // if TRUE, the exit method is called for exiting an instance that is copied afterwards (online change)
END_VAR
// Do Nothing
END_METHOD

(* ---------------------------------------------------------------------------
Func name   : 	FB_init
Description : 	Constructor
Inputs      :	signal	-	Pointer to the output BOOL signal value
Returns     : 	None
Notes       : 	
--------------------------------------------------------------------------- *)

METHOD FB_init : BOOL
VAR_INPUT
	bInitRetains 		: BOOL; 			// if TRUE, the retain variables are initialized (warm start / cold start)
    bInCopyCode  		: BOOL; 			// if TRUE, the instance afterwards gets moved into the copy code (online change)
	signal				: POINTER TO BOOL;	// Pointer to output BOOL signal value 
END_VAR
// Set the local signal pointer
m_signal := signal;
END_METHOD

